// TwinCAT 3 PLC project GW200_plc
// ProgramVersion: 3.1.4024.0
// libraries:
//   Tc2_SerialCom, * (Beckhoff Automation GmbH)
//   Tc2_Standard, * (Beckhoff Automation GmbH)
//   Tc2_System, * (Beckhoff Automation GmbH)
//   Tc2_Utilities, * (Beckhoff Automation GmbH)
//   Tc3_JsonXml, * (Beckhoff Automation GmbH)
//   Tc3_Module, * (Beckhoff Automation GmbH)
// project tree:
//   Base/Alarms/Alarm/ E_ALARM_ACK_TYPE.TcDUT, E_ALARM_STATE.TcDUT, FB_ALARM.TcPOU, TYP_ALARM_CONFIG.TcDUT
//   Base/Alarms/Handler/ FBA_ALARM_HANDLER.TcPOU, FB_ALARM_HANDLER.TcPOU
//   Base/Alarms/ I_ALARM_HANDLER.TcIO, TYP_ALARM_DEVICE_CONFIG.TcDUT
//   Base/Alarms/Repository/ FB_ALARM_INSTANCE.TcPOU, FB_ALARM_REPOSITORY.TcPOU, TYP_ALARM_HISTORY_ENTRY.TcDUT, TYP_VISU_ALARM.TcDUT
//   Base/ BASE.TcPOU
//   Base/Basic/ FB_RS_TRIG.TcPOU
//   Base/DateTime/ FB_DATETIME.TcPOU
//   Base/Files/ FB_FIND_FILES.TcPOU
//   Base/Math/ FC_SCALE.TcPOU, TYP_SCALE_CONF.TcDUT
//   Base/Motion/DC/DcMotor/ FB_DC_MOTOR.TcPOU, TYP_DC_MOTOR_STATUS.TcDUT
//   Base/Motion/DC/DcMotor/Hardware/ TYP_DC_MOTOR_HW.TcDUT, TYP_DC_MOTOR_HW_IN.TcDUT, TYP_DC_MOTOR_HW_OUT.TcDUT
//   Base/Motion/DC/Faulhaber_SC/ FB_FAULHABER_SC.TcPOU, TYP_FAULHABER_SC_CTRL.TcDUT
//   Base/Motion/DC/Faulhaber_SC/Hardware/ TYP_FAULHABER_SC_HW.TcDUT, TYP_FAULHABER_SC_HW_IN.TcDUT, TYP_FAULHABER_SC_HW_OUT.TcDUT
//   Base/Pneumatics/ FB_VALVE_TIMEOUT_ALARM.TcPOU, TYP_VALVE_POS_CONF.TcDUT, TYP_VALVE_POS_HW.TcDUT, TYP_VALVE_TIMEOUT_ALARM_CONF.TcDUT
//   Base/Pneumatics/VacuumGen/ FB_VAC_GEN.TcPOU, TYP_VAC_GEN_ALARM_CONF.TcDUT, TYP_VAC_GEN_CONF.TcDUT, TYP_VAC_GEN_CTRL.TcDUT, TYP_VAC_GEN_STATUS.TcDUT
//   Base/Pneumatics/VacuumGen/Hardware/ TYP_VAC_GEN_HW.TcDUT, TYP_VAC_GEN_HW_IN.TcDUT, TYP_VAC_GEN_HW_OUT.TcDUT
//   Base/Pneumatics/Valve53/ FB_VALVE_53.TcPOU, TYP_VALVE_53_CONF.TcDUT, TYP_VALVE_53_CTRL.TcDUT, TYP_VALVE_53_STATUS.TcDUT
//   Base/Pneumatics/Valve53/Hardware/ TYP_VALVE_53_HW.TcDUT, TYP_VALVE_53_HW_IN.TcDUT, TYP_VALVE_53_HW_OUT.TcDUT
//   Base/Robotics/ TYP_REAL_XYZ.TcDUT
//   Base/Robotics/UR/Profinet/ E_UR_PN_ROBOT_MODE.TcDUT, FB_UR_PN.TcPOU, FB_UR_PN_IO.TcPOU, TYP_HW_UR_PN.TcDUT, TYP_HW_UR_PN_IN.TcDUT, TYP_HW_UR_PN_OUT.TcDUT, TYP_UR_PN_STATE.TcDUT, TYP_UR_PN_TCP.TcDUT
//   Base/Serial/ FB_EL6001_LINE_CTRL.TcPOU, FB_EL6001_RS232.TcPOU, TYP_HW_EL6001.TcDUT, TYP_HW_EL6001_IN.TcDUT, TYP_HW_EL6001_OUT.TcDUT, TYP_SERIAL_DATA.TcDUT
//   Base/Signalling/BannerK50/ FB_BANNER_K50.TcPOU
//   Base/Signalling/BannerK50/Hardware/ TYP_BAN_K50_HW.TcDUT, TYP_BAN_K50_HW_IN.TcDUT, TYP_BAN_K50_HW_OUT.TcDUT
//   Base/Signalling/Lights/ TYP_RYG_TOWER_HW.TcDUT, TYP_RYG_TOWER_HW_OUT.TcDUT
//   Base/Signalling/RGB/ FB_RGB_LED.TcPOU
//   Base/Signalling/RGB/Hardware/ TYP_RGB_LED_CHANNEL.TcDUT, TYP_RGB_LED_CHANNEL_OUT.TcDUT, TYP_RGB_LED_HW.TcDUT
//   Base/States/ FBA_SEQUENCE.TcPOU, FB_SEQUENCE_VISU.TcPOU, FB_STATE_MACHINE.TcPOU
//   Base/String/ FB_STRINGS.TcPOU
//   Base/Tooling/DepragAST11/ TYP_DEPRAG_AST11_HW.TcDUT, TYP_DEPRAG_AST11_HW_IN.TcDUT, TYP_DEPRAG_AST11_HW_OUT.TcDUT
//   Base/Twiddlers/ FC_FLIP_DWORD.TcPOU, FC_FLIP_WORD.TcPOU, FC_GET_BIT_IN_BYTE.TcPOU, FC_MEMCPY_FLIP_WORD.TcPOU, FC_MEMCPY_SWAP_BYTE.TcPOU, FC_MEMCPY_SWAP_WORD.TcPOU, FC_SET_BIT_IN_BYTE.TcPOU
//   Base/Vision/Cognex/3D_L4000/OpcUa/ TYP_HW_L4000_OPC.TcDUT, TYP_HW_L4000_OPC_IN.TcDUT, TYP_HW_L4000_OPC_JOB_CHANGE.TcDUT, TYP_HW_L4000_OPC_JOB_CHANGE_IN.TcDUT, TYP_HW_L4000_OPC_JOB_CHANGE_OUT.TcDUT, TYP_HW_L4000_OPC_OUT.TcDUT
//   Base/Vision/Cognex/3D_L4000/Profinet/ TYP_HW_L4000.TcDUT, TYP_HW_L4000_ACQ_CTRL.TcDUT, TYP_HW_L4000_ACQ_STATUS.TcDUT, TYP_HW_L4000_EXT_CTRL.TcDUT, TYP_HW_L4000_EXT_STATUS.TcDUT, TYP_HW_L4000_IN.TcDUT, TYP_HW_L4000_INSP_CTRL.TcDUT, TYP_HW_L4000_INSP_RESULTS.TcDUT, TYP_HW_L4000_INSP_STATUS.TcDUT, TYP_HW_L4000_OUT.TcDUT
//   Main/ E_MAIN_STATE.TcDUT, E_COLD_START_STATE.TcDUT, MAIN.TcPOU
//   Main/PressureControl/ FB_PRES_CNTRL.TcPOU, gPresCntrl.TcGVL, TYP_PRES_CNTRL_STATUS.TcDUT, TYP_PRES_CNTRL_PARAMETER.TcDUT, TYP_PRES_CNTRL_CONTROL.TcDUT
//   Main/PurgeN2/ E_N2_STATES.TcDUT, FB_N2_DEVICE.TcPOU, FB_PURGE_N2.TcPOU, gPurgeN2.TcGVL, TYP_PURGE_N2_STATUS.TcDUT, TYP_PURGE_N2_PARAMETER.TcDUT, TYP_PURGE_N2_CONTROL.TcDUT
//   / PlcTask.TcTTO
// real-time tasks:
//   TASK PlcTask: cycle T#10ms, priority 20, ADS port 350

CONFIGURATION GW200_plc
    RESOURCE PLC ON TwinCAT3
        TASK PlcTask(INTERVAL := T#10ms, PRIORITY := 20);
        PROGRAM MAIN WITH PlcTask : MAIN;
    END_RESOURCE
END_CONFIGURATION

// ---- Base/Alarms/Alarm/E_ALARM_ACK_TYPE.TcDUT
{attribute 'qualified_only'}
{attribute 'strict'}
TYPE E_ALARM_ACK_TYPE :
(
	ONLY_ACK := 0, // Alarm will clear only after acknowledgement, reset not necessary
	ONLY_RESET := 1, // Alarm will clear only after reset, acknowledgement not necessary
	ACK_AFTER_RESET := 2, // Alarm will clear if acknowledgement is done after reset
	ACK_OR_RESET := 3, // Alarm will clear if reset or acknowledged, whichever comes first
	ACK_AND_RESET := 4 // Alarm will clear if reset and acknowledged, order not important
);
END_TYPE

// ---- Base/Alarms/Alarm/E_ALARM_STATE.TcDUT
{attribute 'qualified_only'}
{attribute 'strict'}
{attribute 'to_string'}
TYPE E_ALARM_STATE :
(
	INACTIVE := 0,
	ACTIVE_UNACK := 1,
	ACTIVE_ACK := 2,
	INACTIVE_UNACK := 4
);
END_TYPE

// ---- Base/Alarms/Alarm/TYP_ALARM_CONFIG.TcDUT
TYPE TYP_ALARM_CONFIG :
STRUCT
	Name : STRING;
	Priority : INT;
	Code : DINT;
	Acknowledge : E_ALARM_ACK_TYPE;
	MultiInstance : BOOL; // Alarm going active again creates new alarm instance
END_STRUCT
END_TYPE

// ---- Base/Alarms/Repository/TYP_ALARM_HISTORY_ENTRY.TcDUT
TYPE TYP_ALARM_HISTORY_ENTRY :
STRUCT
	Timestamp : DT;
	Name : STRING;
	Message : STRING;
	PreviousState : STRING;
	NewState : STRING;
	Code : DINT;
	Priority : INT;
END_STRUCT
END_TYPE

// ---- Base/Alarms/Repository/TYP_VISU_ALARM.TcDUT
TYPE TYP_VISU_ALARM :
STRUCT
	Timestamp : DT;
	Name : STRING;
	Message : STRING;
	State : STRING;
	Code : DINT;
	Priority : INT;
END_STRUCT
END_TYPE

// ---- Base/Alarms/TYP_ALARM_DEVICE_CONFIG.TcDUT
TYPE TYP_ALARM_DEVICE_CONFIG :
STRUCT
	Name : STRING;
	Handler : REFERENCE TO FB_ALARM_HANDLER;
END_STRUCT
END_TYPE

// ---- Base/Math/TYP_SCALE_CONF.TcDUT
TYPE TYP_SCALE_CONF :
STRUCT
	InMin : REAL;
	InMax : REAL;
	OutMin : REAL;
	OutMax : REAL;
END_STRUCT
END_TYPE

// ---- Base/Motion/DC/DcMotor/Hardware/TYP_DC_MOTOR_HW.TcDUT
TYPE TYP_DC_MOTOR_HW :
STRUCT
	In : TYP_DC_MOTOR_HW_IN;
	Out : TYP_DC_MOTOR_HW_OUT;
END_STRUCT
END_TYPE

// ---- Base/Motion/DC/DcMotor/Hardware/TYP_DC_MOTOR_HW_IN.TcDUT
TYPE TYP_DC_MOTOR_HW_IN :
STRUCT
	LimitHP AT %I* : BOOL;
	LimitWP AT %I* : BOOL;
END_STRUCT
END_TYPE

// ---- Base/Motion/DC/DcMotor/Hardware/TYP_DC_MOTOR_HW_OUT.TcDUT
TYPE TYP_DC_MOTOR_HW_OUT :
STRUCT
	Direction AT %Q* : BOOL;
	Run AT %Q* : BOOL;
END_STRUCT
END_TYPE

// ---- Base/Motion/DC/DcMotor/TYP_DC_MOTOR_STATUS.TcDUT
TYPE TYP_DC_MOTOR_STATUS :
STRUCT
	ReachedHP : BOOL;
	ReachedWP : BOOL;
END_STRUCT
END_TYPE

// ---- Base/Motion/DC/Faulhaber_SC/Hardware/TYP_FAULHABER_SC_HW.TcDUT
TYPE TYP_FAULHABER_SC_HW :
STRUCT
	In : TYP_FAULHABER_SC_HW_IN;
	Out : TYP_FAULHABER_SC_HW_OUT;
END_STRUCT
END_TYPE

// ---- Base/Motion/DC/Faulhaber_SC/Hardware/TYP_FAULHABER_SC_HW_IN.TcDUT
TYPE TYP_FAULHABER_SC_HW_IN :
STRUCT
	Fault AT %I*: BOOL;
END_STRUCT
END_TYPE

// ---- Base/Motion/DC/Faulhaber_SC/Hardware/TYP_FAULHABER_SC_HW_OUT.TcDUT
TYPE TYP_FAULHABER_SC_HW_OUT :
STRUCT
	Speed AT %Q*: INT;
	Direction AT %Q*: BOOL;
END_STRUCT
END_TYPE

// ---- Base/Motion/DC/Faulhaber_SC/TYP_FAULHABER_SC_CTRL.TcDUT
TYPE TYP_FAULHABER_SC_CTRL :
STRUCT	
	Enable : BOOL; // Enable action
	Run : BOOL; // Run motor
	Speed : INT; // Setpoint speed
END_STRUCT
END_TYPE

// ---- Base/Pneumatics/TYP_VALVE_POS_CONF.TcDUT
TYPE TYP_VALVE_POS_CONF :
STRUCT
	Sensorless : BOOL; (* no sensor, reached status after SensorlessDelay *)
	SensorlessDelay : TIME; (* delay for reached status in sensorless mode *)
	Permanent : BOOL := TRUE; // Output stays on after reaching position
	Timeout : TYP_VALVE_TIMEOUT_ALARM_CONF;
END_STRUCT
END_TYPE

// ---- Base/Pneumatics/TYP_VALVE_POS_HW.TcDUT
TYPE TYP_VALVE_POS_HW :
STRUCT
	ReachedHP AT %I* : BOOL;
	ReachedWP AT %I* : BOOL;
END_STRUCT
END_TYPE

// ---- Base/Pneumatics/TYP_VALVE_TIMEOUT_ALARM_CONF.TcDUT
TYPE TYP_VALVE_TIMEOUT_ALARM_CONF :
STRUCT
	Enable : BOOL := TRUE; // Alarm enabled
	Delay : TIME := T#10S; // Delay before alarm is activated
END_STRUCT
END_TYPE

// ---- Base/Pneumatics/VacuumGen/Hardware/TYP_VAC_GEN_HW.TcDUT
TYPE TYP_VAC_GEN_HW :
STRUCT
	In : TYP_VAC_GEN_HW_IN;
	Out : TYP_VAC_GEN_HW_OUT;
END_STRUCT
END_TYPE

// ---- Base/Pneumatics/VacuumGen/Hardware/TYP_VAC_GEN_HW_IN.TcDUT
TYPE TYP_VAC_GEN_HW_IN :
STRUCT
	ReachedVac AT %I* : BOOL;
END_STRUCT
END_TYPE

// ---- Base/Pneumatics/VacuumGen/Hardware/TYP_VAC_GEN_HW_OUT.TcDUT
TYPE TYP_VAC_GEN_HW_OUT :
STRUCT
	EnableVac AT %Q* : BOOL;
	ReleaseVac AT %Q* : BOOL;
END_STRUCT
END_TYPE

// ---- Base/Pneumatics/VacuumGen/TYP_VAC_GEN_ALARM_CONF.TcDUT
TYPE TYP_VAC_GEN_ALARM_CONF :
STRUCT
	Enable : BOOL := TRUE;
	Timeout : TIME := T#4S;
END_STRUCT
END_TYPE

// ---- Base/Pneumatics/VacuumGen/TYP_VAC_GEN_CONF.TcDUT
TYPE TYP_VAC_GEN_CONF :
STRUCT
	Permanent : BOOL := TRUE; // Holds output even after reaching vacuum
	Alarm : TYP_VAC_GEN_ALARM_CONF;
END_STRUCT
END_TYPE

// ---- Base/Pneumatics/VacuumGen/TYP_VAC_GEN_CTRL.TcDUT
TYPE TYP_VAC_GEN_CTRL :
STRUCT
	Enable : BOOL := TRUE; // Enable vacuum gen control
	EnableActivate : BOOL := TRUE; // Enable vacuum activation
	EnableRelease : BOOL := TRUE; // Enable release activation
	ServiceEnable : BOOL;
	ServiceActivate : BOOL;
	ServiceRelease : BOOL;
END_STRUCT
END_TYPE

// ---- Base/Pneumatics/VacuumGen/TYP_VAC_GEN_STATUS.TcDUT
TYPE TYP_VAC_GEN_STATUS :
STRUCT
	ReachedVac : BOOL;
	Error : BOOL;
END_STRUCT
END_TYPE

// ---- Base/Pneumatics/Valve53/Hardware/TYP_VALVE_53_HW.TcDUT
TYPE TYP_VALVE_53_HW :
STRUCT
	In : TYP_VALVE_53_HW_IN;
	Out : TYP_VALVE_53_HW_OUT;
END_STRUCT
END_TYPE

// ---- Base/Pneumatics/Valve53/Hardware/TYP_VALVE_53_HW_IN.TcDUT
TYPE TYP_VALVE_53_HW_IN :
STRUCT
	ReachedHP AT %I* : BOOL;
	ReachedWP AT %I* : BOOL;
END_STRUCT
END_TYPE

// ---- Base/Pneumatics/Valve53/Hardware/TYP_VALVE_53_HW_OUT.TcDUT
TYPE TYP_VALVE_53_HW_OUT :
STRUCT
	CmdHP AT %Q* : BOOL;
	CmdWP AT %Q* : BOOL;
END_STRUCT
END_TYPE

// ---- Base/Pneumatics/Valve53/TYP_VALVE_53_CONF.TcDUT
TYPE TYP_VALVE_53_CONF :
STRUCT
	HP : TYP_VALVE_POS_CONF;
	WP : TYP_VALVE_POS_CONF;
	HP_WP : TYP_VALVE_TIMEOUT_ALARM_CONF; // Alarm for both HP and WP sensors active
END_STRUCT
END_TYPE

// ---- Base/Pneumatics/Valve53/TYP_VALVE_53_CTRL.TcDUT
TYPE TYP_VALVE_53_CTRL :
STRUCT
	Enable : BOOL := TRUE; (* Enable movement in auto mode *)
	EnableHP : BOOL := TRUE; (* Allow movement to HP *)
	EnableWP : BOOL := TRUE; (* Allow movement to WP *)
	ServiceEnable : BOOL; (* Enable movement in Service Mode NB!! This ignores all other enable/disable commands *)
	ServiceHP : BOOL; (* Command movement to Home Position NB!! This ignores all other enable/disable commands *)
	ServiceWP : BOOL; (* Command movement to Wome Position NB!! This ignores all other enable/disable commands *)
	BlockOutputs : BOOL; // Do not allow to switch outputs
END_STRUCT
END_TYPE

// ---- Base/Pneumatics/Valve53/TYP_VALVE_53_STATUS.TcDUT
TYPE TYP_VALVE_53_STATUS :
STRUCT
	ReachedHP : BOOL;
	ReachedWP : BOOL;
	Error : BOOL;
END_STRUCT
END_TYPE

// ---- Base/Robotics/TYP_REAL_XYZ.TcDUT
TYPE TYP_REAL_XYZ :
STRUCT
	X : REAL;
	Y : REAL;
	Z : REAL;
END_STRUCT
END_TYPE

// ---- Base/Robotics/UR/Profinet/E_UR_PN_ROBOT_MODE.TcDUT
{attribute 'qualified_only'}
//{attribute 'strict'}
{attribute 'to_string'}
TYPE E_UR_PN_ROBOT_MODE :
(
	DISCONNECTED := 0,
	CONFIRM_SAFETY := 1,
	BOOTING := 2,
	POWER_OFF := 3,
	POWER_ON := 4,
	IDLE := 5,
	BACKDRIVE := 6,
	RUNNING := 7
);
END_TYPE

// ---- Base/Robotics/UR/Profinet/TYP_HW_UR_PN.TcDUT
TYPE TYP_HW_UR_PN :
STRUCT
	In : TYP_HW_UR_PN_IN;
	Out : TYP_HW_UR_PN_OUT;
END_STRUCT
END_TYPE

// ---- Base/Robotics/UR/Profinet/TYP_HW_UR_PN_IN.TcDUT
TYPE TYP_HW_UR_PN_IN :
STRUCT
	T2OURState AT %I*: ARRAY[0..31] OF BYTE;
	T2OURIO AT %I*: ARRAY[0..67] OF BYTE;
	T2OURJoints AT %I*: ARRAY[0..103] OF BYTE;
	T2OURTCP AT %I*: ARRAY[0..75] OF BYTE;
	T2OURBitReg AT %I*: ARRAY[0..7] OF BYTE;
	T2OURIntReg AT %I*: ARRAY[0..95] OF BYTE;
	T2OURFloatReg AT %I*: ARRAY[0..95] OF BYTE;
END_STRUCT
END_TYPE

// ---- Base/Robotics/UR/Profinet/TYP_HW_UR_PN_OUT.TcDUT
TYPE TYP_HW_UR_PN_OUT :
STRUCT
	O2TURIO AT %Q*: ARRAY[0..23] OF BYTE;
	O2TURGenReg1 AT %Q*: ARRAY[0..99] OF BYTE;
	O2TURGenReg2 AT %Q*: ARRAY[0..99] OF BYTE;
END_STRUCT
END_TYPE

// ---- Base/Robotics/UR/Profinet/TYP_UR_PN_STATE.TcDUT
TYPE TYP_UR_PN_STATE :
STRUCT
	MajVersion : USINT; // Controller major version
	MinVersion : USINT; // Controller minor version
	RobotMode : E_UR_PN_ROBOT_MODE;
	RTMd : UINT; // Real time machine days
	RTMh : UINT; // Real time machine hours
	RTMm : UINT; // Real time machine days
	RTMs : UINT; // Real time machine days
	RTMms : UINT; // Real time machine milliseconds
	Power : BOOL;
	ProgramRunning : BOOL;
	PowerButton : BOOL;
	TeachButton : BOOL;
	RobotCurrent : REAL; // Current power consumption A
	NormalMode: BOOL;
	ReducedMode: BOOL;
	ProtectiveStopped: BOOL;
	RecoveryMode: BOOL;
	SafeguardStop: BOOL;
	SystemEmergencyStopped: BOOL;
	RobotEmergencyStopped: BOOL;
	EmergencyStopped: BOOL;
	Violation: BOOL;
	Faulted: BOOL;
	SafetyStopped: BOOL;
END_STRUCT
END_TYPE

// ---- Base/Robotics/UR/Profinet/TYP_UR_PN_TCP.TcDUT
TYPE TYP_UR_PN_TCP :
STRUCT
	Position : TYP_REAL_XYZ;
	PositionR : TYP_REAL_XYZ;
	Velocity : TYP_REAL_XYZ;
	VelocityR : TYP_REAL_XYZ;
	Force : TYP_REAL_XYZ;
	Torque : TYP_REAL_XYZ;
	ForceScalar : REAL;
END_STRUCT
END_TYPE

// ---- Base/Serial/TYP_HW_EL6001.TcDUT
TYPE TYP_HW_EL6001 :
STRUCT
	In : TYP_HW_EL6001_IN;
	Out : TYP_HW_EL6001_OUT;
END_STRUCT
END_TYPE

// ---- Base/Serial/TYP_HW_EL6001_IN.TcDUT
TYPE TYP_HW_EL6001_IN :
STRUCT
	COM AT %I*: KL6InData22B;
END_STRUCT
END_TYPE

// ---- Base/Serial/TYP_HW_EL6001_OUT.TcDUT
TYPE TYP_HW_EL6001_OUT :
STRUCT
	COM AT %Q* : KL6OutData22B;
END_STRUCT
END_TYPE

// ---- Base/Serial/TYP_SERIAL_DATA.TcDUT
TYPE TYP_SERIAL_DATA :
STRUCT
	RxData : COMbuffer;
	TxData : COMbuffer;
END_STRUCT
END_TYPE

// ---- Base/Signalling/BannerK50/Hardware/TYP_BAN_K50_HW.TcDUT
TYPE TYP_BAN_K50_HW :
STRUCT
	In : TYP_BAN_K50_HW_IN;
	Out : TYP_BAN_K50_HW_OUT;
END_STRUCT
END_TYPE

// ---- Base/Signalling/BannerK50/Hardware/TYP_BAN_K50_HW_IN.TcDUT
TYPE TYP_BAN_K50_HW_IN :
STRUCT
	ButtonPressed AT %I* : BOOL;
END_STRUCT
END_TYPE

// ---- Base/Signalling/BannerK50/Hardware/TYP_BAN_K50_HW_OUT.TcDUT
TYPE TYP_BAN_K50_HW_OUT :
STRUCT
	Red AT %Q* : BOOL;
	Yellow AT %Q* : BOOL;
	Green AT %Q* : BOOL;
END_STRUCT
END_TYPE

// ---- Base/Signalling/Lights/TYP_RYG_TOWER_HW.TcDUT
TYPE TYP_RYG_TOWER_HW :
STRUCT
	Out : TYP_RYG_TOWER_HW_OUT;
END_STRUCT
END_TYPE

// ---- Base/Signalling/Lights/TYP_RYG_TOWER_HW_OUT.TcDUT
TYPE TYP_RYG_TOWER_HW_OUT :
STRUCT
	Red AT %Q* : BOOL;
	Yellow AT %Q* : BOOL;
	Green AT %Q* : BOOL;
END_STRUCT
END_TYPE

// ---- Base/Signalling/RGB/Hardware/TYP_RGB_LED_CHANNEL.TcDUT
TYPE TYP_RGB_LED_CHANNEL :
STRUCT
	Out : TYP_RGB_LED_CHANNEL_OUT;
END_STRUCT
END_TYPE

// ---- Base/Signalling/RGB/Hardware/TYP_RGB_LED_CHANNEL_OUT.TcDUT
TYPE TYP_RGB_LED_CHANNEL_OUT :
STRUCT
	PWM AT %Q* : INT;
END_STRUCT
END_TYPE

// ---- Base/Signalling/RGB/Hardware/TYP_RGB_LED_HW.TcDUT
TYPE TYP_RGB_LED_HW :
STRUCT
	Red : TYP_RGB_LED_CHANNEL;
	Green : TYP_RGB_LED_CHANNEL;
	Blue : TYP_RGB_LED_CHANNEL;
END_STRUCT
END_TYPE

// ---- Base/Tooling/DepragAST11/TYP_DEPRAG_AST11_HW.TcDUT
TYPE TYP_DEPRAG_AST11_HW :
STRUCT
	In : TYP_DEPRAG_AST11_HW_IN;
	Out : TYP_DEPRAG_AST11_HW_OUT;
END_STRUCT
END_TYPE

// ---- Base/Tooling/DepragAST11/TYP_DEPRAG_AST11_HW_IN.TcDUT
TYPE TYP_DEPRAG_AST11_HW_IN :
STRUCT
	Ready AT %I*: BOOL;
	OK AT %I*: BOOL;
	NOK AT %I*: BOOL;
END_STRUCT
END_TYPE

// ---- Base/Tooling/DepragAST11/TYP_DEPRAG_AST11_HW_OUT.TcDUT
TYPE TYP_DEPRAG_AST11_HW_OUT :
STRUCT
	Start AT %Q*: BOOL;
END_STRUCT
END_TYPE

// ---- Base/Vision/Cognex/3D_L4000/OpcUa/TYP_HW_L4000_OPC.TcDUT
TYPE TYP_HW_L4000_OPC :
STRUCT
	LoadJob : TYP_HW_L4000_OPC_JOB_CHANGE;
	In : TYP_HW_L4000_OPC_IN;
	Out : TYP_HW_L4000_OPC_OUT;
END_STRUCT
END_TYPE

// ---- Base/Vision/Cognex/3D_L4000/OpcUa/TYP_HW_L4000_OPC_IN.TcDUT
TYPE TYP_HW_L4000_OPC_IN :
STRUCT
	Result AT %I* : ARRAY[1..43] OF REAL;
	Online AT %I* : BOOL;
	ActiveJob AT %I* : STRING;
END_STRUCT
END_TYPE

// ---- Base/Vision/Cognex/3D_L4000/OpcUa/TYP_HW_L4000_OPC_JOB_CHANGE.TcDUT
TYPE TYP_HW_L4000_OPC_JOB_CHANGE :
STRUCT
	In : TYP_HW_L4000_OPC_JOB_CHANGE_IN;
	Out : TYP_HW_L4000_OPC_JOB_CHANGE_OUT;
END_STRUCT
END_TYPE

// ---- Base/Vision/Cognex/3D_L4000/OpcUa/TYP_HW_L4000_OPC_JOB_CHANGE_IN.TcDUT
TYPE TYP_HW_L4000_OPC_JOB_CHANGE_IN :
STRUCT
	ErrorID AT %I* : DINT;
	Done AT %I* : BOOL;
	Busy AT %I* : BOOL;
	Error AT %I* : BOOL;
END_STRUCT
END_TYPE

// ---- Base/Vision/Cognex/3D_L4000/OpcUa/TYP_HW_L4000_OPC_JOB_CHANGE_OUT.TcDUT
TYPE TYP_HW_L4000_OPC_JOB_CHANGE_OUT :
STRUCT
	Execute AT %Q* : BOOL;
	Filename AT %Q* : STRING;
END_STRUCT
END_TYPE

// ---- Base/Vision/Cognex/3D_L4000/OpcUa/TYP_HW_L4000_OPC_OUT.TcDUT
TYPE TYP_HW_L4000_OPC_OUT :
STRUCT
	WriteEnable AT %Q* : BOOL;
	Online AT %Q* : BOOL;
END_STRUCT
END_TYPE

// ---- Base/Vision/Cognex/3D_L4000/Profinet/TYP_HW_L4000.TcDUT
TYPE TYP_HW_L4000 :
STRUCT
	In : TYP_HW_L4000_IN;
	Out : TYP_HW_L4000_OUT;
END_STRUCT
END_TYPE

// ---- Base/Vision/Cognex/3D_L4000/Profinet/TYP_HW_L4000_ACQ_CTRL.TcDUT
TYPE TYP_HW_L4000_ACQ_CTRL :
STRUCT
	AcqTriggerEnable AT %Q* : BOOL;
	AcqTrigger AT %Q* : BOOL;
	ClearExposureComplete AT %Q* : BOOL;
	SetPauseOfOnline AT %Q* : BOOL;
END_STRUCT
END_TYPE

// ---- Base/Vision/Cognex/3D_L4000/Profinet/TYP_HW_L4000_ACQ_STATUS.TcDUT
TYPE TYP_HW_L4000_ACQ_STATUS :
STRUCT
	AcqTriggerReady AT %I* : BOOL;
	AcqTriggerAcknowledge AT %I* : BOOL;
	ExposureComplete AT %I* : BOOL;
	AcqError AT %I* : BOOL;
	Paused AT %I* : BOOL;
	Online AT %I* : BOOL;
	AcqID AT %I* : UINT;
END_STRUCT
END_TYPE

// ---- Base/Vision/Cognex/3D_L4000/Profinet/TYP_HW_L4000_EXT_CTRL.TcDUT
TYPE TYP_HW_L4000_EXT_CTRL :
STRUCT
	Trigger AT %Q* : ARRAY[0..7] OF BOOL;
END_STRUCT
END_TYPE

// ---- Base/Vision/Cognex/3D_L4000/Profinet/TYP_HW_L4000_EXT_STATUS.TcDUT
TYPE TYP_HW_L4000_EXT_STATUS :
STRUCT
	Acknowledge AT %I* : ARRAY[0..7] OF BOOL;
END_STRUCT
END_TYPE

// ---- Base/Vision/Cognex/3D_L4000/Profinet/TYP_HW_L4000_IN.TcDUT
TYPE TYP_HW_L4000_IN :
STRUCT
	AcqStatus : TYP_HW_L4000_ACQ_STATUS;
	InspStatus : TYP_HW_L4000_INSP_STATUS;
	CommandResult AT %I* : UINT;
	ExternalEvent : TYP_HW_L4000_EXT_STATUS;
	InspResults : TYP_HW_L4000_INSP_RESULTS;
END_STRUCT
END_TYPE

// ---- Base/Vision/Cognex/3D_L4000/Profinet/TYP_HW_L4000_INSP_CTRL.TcDUT
TYPE TYP_HW_L4000_INSP_CTRL :
STRUCT
	EnableResultsBuffering AT %Q* : BOOL;
	AckInspectionResults AT %Q* : BOOL;
	SetUserData AT %Q* : BOOL;
	ExecuteCommand AT %Q* : BOOL;
	ClearError AT %Q* : BOOL;
END_STRUCT
END_TYPE

// ---- Base/Vision/Cognex/3D_L4000/Profinet/TYP_HW_L4000_INSP_RESULTS.TcDUT
TYPE TYP_HW_L4000_INSP_RESULTS :
STRUCT
	InspectionID AT %I* : UINT;
	InspectionResultCode AT %I* : UINT;
	Results AT %I* : ARRAY[0..63] OF BYTE;
END_STRUCT
END_TYPE

// ---- Base/Vision/Cognex/3D_L4000/Profinet/TYP_HW_L4000_INSP_STATUS.TcDUT
TYPE TYP_HW_L4000_INSP_STATUS :
STRUCT
	SystemReady AT %I* : BOOL;
	InspectionCompleted AT %I* : BOOL;
	ResultsBufferOverrun AT %I* : BOOL;
	ResultsValid AT %I* : BOOL;
	CommandExecuting AT %I* : BOOL;
	CommandCompleted AT %I* : BOOL;
	CommandFailed AT %I* : BOOL;
	SetUserDataAcknowledge AT %I* : BOOL;
	ResultsPassed AT %I* : BOOL;
	Error AT %I* : BOOL;
	ErrorID AT %I* : UINT;
END_STRUCT
END_TYPE

// ---- Base/Vision/Cognex/3D_L4000/Profinet/TYP_HW_L4000_OUT.TcDUT
TYPE TYP_HW_L4000_OUT :
STRUCT
	AcqCtrl : TYP_HW_L4000_ACQ_CTRL;
	InspCtrl : TYP_HW_L4000_INSP_CTRL;
	CommandID AT %Q* : UINT;
	ExternalEvent : TYP_HW_L4000_EXT_CTRL;
	UserData AT %Q* : ARRAY[0..63] OF BYTE;
END_STRUCT
END_TYPE

// ---- Main/E_MAIN_STATE.TcDUT
{attribute 'qualified_only'}
{attribute 'strict'}
TYPE E_MAIN_STATE :
(
	NULL := 0,
	IDLE,
	COLD_START,
	HOT_START,
	SHUT_DOWN,
	PRODUCTION,
	HOT_STANDBY,
	COLD_STANDBY
);
END_TYPE

// ---- Main/E_COLD_START_STATE.TcDUT
{attribute 'qualified_only'}
{attribute 'strict'}
TYPE E_COLD_START_STATE :
(
	NULL := 0,
	N2_PURGE,
	TEMPERATURE,	
	PRESSURISE,
	H2_PURGE
);
END_TYPE

// ---- Main/PressureControl/TYP_PRES_CNTRL_STATUS.TcDUT
TYPE TYP_PRES_CNTRL_STATUS :
STRUCT
	Done : BOOL;
	Executing: BOOL;
	Error : BOOL;
END_STRUCT
END_TYPE

// ---- Main/PressureControl/TYP_PRES_CNTRL_PARAMETER.TcDUT
TYPE TYP_PRES_CNTRL_PARAMETER :
STRUCT
	SetPoint : REAL;
END_STRUCT
END_TYPE

// ---- Main/PressureControl/TYP_PRES_CNTRL_CONTROL.TcDUT
TYPE TYP_PRES_CNTRL_CONTROL :
STRUCT
	Execute : BOOL;
END_STRUCT
END_TYPE

// ---- Main/PurgeN2/E_N2_STATES.TcDUT
{attribute 'qualified_only'}
{attribute 'strict'}
TYPE E_N2_STATES :
(
	STATE1,
	STATE2,
	STATE3
);
END_TYPE

// ---- Main/PurgeN2/TYP_PURGE_N2_STATUS.TcDUT
TYPE TYP_PURGE_N2_STATUS :
STRUCT
	Done : BOOL;
	Executing: BOOL;
	Error : BOOL;
END_STRUCT
END_TYPE

// ---- Main/PurgeN2/TYP_PURGE_N2_PARAMETER.TcDUT
TYPE TYP_PURGE_N2_PARAMETER :
STRUCT
	NoPurge : INT;
END_STRUCT
END_TYPE

// ---- Main/PurgeN2/TYP_PURGE_N2_CONTROL.TcDUT
TYPE TYP_PURGE_N2_CONTROL :
STRUCT
	Execute : BOOL;
END_STRUCT
END_TYPE

// ---- Main/PressureControl/gPresCntrl.TcGVL
{attribute 'qualified_only'}
VAR_GLOBAL
	Control : TYP_PRES_CNTRL_CONTROL;
	Parameter : TYP_PRES_CNTRL_PARAMETER;
	Status : TYP_PRES_CNTRL_STATUS;
END_VAR

// ---- Main/PurgeN2/gPurgeN2.TcGVL
{attribute 'qualified_only'}
VAR_GLOBAL
	Control: TYP_PURGE_N2_CONTROL;
	Parameter : TYP_PURGE_N2_PARAMETER;
	Status : TYP_PURGE_N2_STATUS;
END_VAR

// ---- Base/Alarms/I_ALARM_HANDLER.TcIO
INTERFACE I_ALARM_HANDLER

METHOD RegisterAlarm : REFERENCE TO FBA_ALARM_HANDLER
VAR_INPUT
	Alarm : REFERENCE TO FB_ALARM;
	Prefix : STRING := '';
	Update : BOOL := TRUE;
END_VAR
END_METHOD

END_INTERFACE

// ---- Main/MAIN.TcPOU
PROGRAM MAIN
VAR
	//State machines
	fbMainState : FB_STATE_MACHINE;
	fbColdStartState : FB_STATE_MACHINE;
	eMainState : E_MAIN_STATE;
	eColdStartState : E_COLD_START_STATE;
	//Alarm handler
	fbAlarmRepository : FB_ALARM_REPOSITORY;
	fbMainHandler : FB_ALARM_HANDLER;
	fbColdStartHandler : FB_ALARM_HANDLER;
	fbAlarms : ARRAY[0..99] OF FB_ALARM_INSTANCE;
	fbVisuAlarms : ARRAY[0..99] OF TYP_VISU_ALARM;
	fbEmStopAlarm : FB_ALARM;
	//Control loops and function blocks
	fbPurgeN2 : FB_PURGE_N2;
	fbPresCntrl : FB_PRES_CNTRL;
	
	bTestalarm : BOOL;
	bTestReset : BOOL;
	bTestAcknowledge : BOOL;
	
	getZone : FB_LocalSystemTime;
END_VAR

//Alarm function blocks
fbAlarmRepository(Alarms := fbAlarms, VisuAlarms := fbVisuAlarms);
fbMainHandler(Prefix := 'MAIN', Repository := fbAlarmRepository);
fbColdStartHandler(Prefix := 'COLD_START', Repository := fbAlarmRepository);

fbEmStopAlarm.Config.Acknowledge := E_ALARM_ACK_TYPE.ACK_AND_RESET;
fbEmStopAlarm.Config.Name := 'EMERGENCY_STOP_ACTIVATED';
fbEmStopAlarm.Config.Priority := 3;
fbEmStopAlarm.Config.Code := 0001;
fbEmStopAlarm(Handler := fbMainHandler);

//Control loops, control functionblocks
fbPurgeN2(AlarmRepository := fbAlarmRepository, Control := gPurgeN2.Control, Parameter := gPurgeN2.Parameter, Status => gPurgeN2.Status);
fbPresCntrl(Control := gPresCntrl.Control, Parameter := gPresCntrl.Parameter, Status => gPresCntrl.Status);

//Example how alarms work
IF bTestalarm THEN
	fbEmStopAlarm.Activate();
ELSIF bTestReset THEN
	fbEmStopAlarm.Reset();
ELSIF bTestAcknowledge THEN
	fbEmStopAlarm.Acknowledge();
END_IF

CASE fbMainState.CurrentState OF //Main state machine
	E_MAIN_STATE.IDLE:
	 //
	E_MAIN_STATE.COLD_START: //Cold start state
		CASE fbColdStartState.CurrentState OF
			E_COLD_START_STATE.N2_PURGE: //Nitorgen purge state
				IF fbColdStartState._firstCycle THEN
					gPurgeN2.Parameter.NoPurge := 5;
					gPurgeN2.Control.Execute := TRUE;
					gPresCntrl.Parameter.SetPoint := 2.0;
					gPresCntrl.Control.Execute := TRUE;
				ELSIF NOT fbColdStartState.ChangePending THEN
					IF gPurgeN2.Status.Done THEN
						fbColdStartState.ChangeState(E_COLD_START_STATE.TEMPERATURE);
					END_IF
				END_IF	
			E_COLD_START_STATE.TEMPERATURE:
				//
			E_COLD_START_STATE.PRESSURISE:
				//
			E_COLD_START_STATE.H2_PURGE:
				//
		END_CASE	
	
	E_MAIN_STATE.HOT_STANDBY:
		//
	E_MAIN_STATE.PRODUCTION:
		//
	E_MAIN_STATE.COLD_STANDBY:
		//
	E_MAIN_STATE.HOT_START:
		//
	E_MAIN_STATE.SHUT_DOWN:
		//
END_CASE

getZone();

fbMainState(State := eMainState, AlarmHandler := fbMainHandler, StateAsString := TO_STRING(eMainState));
fbColdStartState(State := eColdStartState, AlarmHandler := fbColdStartHandler, StateAsString := TO_STRING(eColdStartState));

END_PROGRAM

// ---- Base/States/FB_STATE_MACHINE.TcPOU
FUNCTION_BLOCK FB_STATE_MACHINE
VAR_IN_OUT
	State : INT;
	AlarmHandler : FB_ALARM_HANDLER;
END_VAR
VAR_INPUT
	StateAsString : STRING;
	DebugMode : BOOL;
	DebugNext : BOOL;
	StopAllowed : BOOL;
	Timeout : TIME;
END_VAR
VAR_OUTPUT
	CurrentState : INT;
	_firstCycle : BOOL := TRUE;
	StateChangeTime : TIME := TIME();
	Running : BOOL;
	Stopped : BOOL;
	StopRequested : BOOL;
	PreviousState : INT;
END_VAR
VAR
	_changePending : BOOL;
	DelayStart : TIME;
	ChangeDelay : TIME;
	NewState : INT;
	NextState : INT;
	TimeoutAlarm : FB_ALARM;
END_VAR

IF NOT DebugMode THEN
	DebugNext := FALSE;
END_IF;

IF Running AND StopRequested AND StopAllowed THEN
	Running := FALSE;
	Stopped := TRUE;
	StopRequested := FALSE;
END_IF;

IF NewState <> CurrentState AND (NOT DebugMode OR DebugNext) AND Running THEN
	PreviousState := CurrentState;
	CurrentState := NewState;
	StateChangeTime := TIME();
	_firstCycle := TRUE;
	DebugNext := FALSE;
	
	Timeout := T#0S;
	DelayStart := T#0S;
	ChangeDelay := T#0S;
	_changePending := FALSE;
	NextState := 0;
ELSE
	_firstCycle := FALSE;
END_IF;

IF _changePending AND TIME() >= (DelayStart + ChangeDelay) THEN
	THIS^.NewState := NextState;
END_IF;

IF Timeout > T#0S AND THIS^.GetElapsedTime() > Timeout  THEN
	IF NOT TimeoutAlarm.IsActive THEN
		TimeoutAlarm.Config.Name := CONCAT(StateAsString, '*TIMEOUT_ALARM');
		TimeoutAlarm.Activate();
	END_IF;
END_IF;

TimeoutAlarm.Config.Acknowledge := E_ALARM_ACK_TYPE.ONLY_ACK;
TimeoutAlarm.Config.MultiInstance := TRUE;
TimeoutAlarm(Handler := AlarmHandler);

State := CurrentState;

StopAllowed := FALSE;

PROPERTY PUBLIC ChangePending : BOOL
GET
ChangePending := THIS^._changePending;
END_GET
END_PROPERTY

METHOD ChangeState : REFERENCE TO FB_STATE_MACHINE
VAR_INPUT
	State : INT;
END_VAR
IF NOT _changePending AND THIS^.Running THEN
	_changePending := TRUE;
	NextState := State;
END_IF;

ChangeState REF= THIS^;
END_METHOD

METHOD ChangeStateAfterDelay : REFERENCE TO FB_STATE_MACHINE
VAR_INPUT
	State : INT;
	Delay : TIME;
END_VAR
IF NOT _changePending AND THIS^.Running THEN
	_changePending := TRUE;
	NextState := State;
	DelayStart := TIME();
	ChangeDelay := Delay;
END_IF;

ChangeStateAfterDelay REF= THIS^;
END_METHOD

PROPERTY PUBLIC FirstCycle : BOOL
GET
FirstCycle := _firstCycle AND Running;
END_GET
END_PROPERTY

METHOD PUBLIC GetElapsedTime : TIME
VAR_INPUT
END_VAR
GetElapsedTime := TIME() - StateChangeTime;
END_METHOD

METHOD PUBLIC Reset : REFERENCE TO FB_STATE_MACHINE
VAR_INPUT
END_VAR
THIS^.CurrentState := 0;
THIS^.NewState := 0;
THIS^._firstCycle := TRUE;
THIS^.StateChangeTime := TIME();
THIS^._changePending := FALSE;
THIS^.DelayStart := T#0S;
THIS^.ChangeDelay := T#0S;
THIS^.NextState := 0;
THIS^.Running := FALSE;
THIS^.Stopped := FALSE;
THIS^.StopRequested := FALSE;

Reset REF= THIS^;
END_METHOD

{attribute 'TcRpcEnable'}
METHOD PUBLIC Start : REFERENCE TO FB_STATE_MACHINE
VAR_INPUT
END_VAR
THIS^.Running := TRUE;
THIS^.StopRequested := FALSE;

Start REF= THIS^;
END_METHOD

{attribute 'TcRpcEnable'}
METHOD PUBLIC Stop : REFERENCE TO FB_STATE_MACHINE
VAR_INPUT
END_VAR
THIS^.StopRequested := TRUE;

Stop REF= THIS^;
END_METHOD

END_FUNCTION_BLOCK

// ---- Base/Alarms/Handler/FB_ALARM_HANDLER.TcPOU
FUNCTION_BLOCK PUBLIC FB_ALARM_HANDLER EXTENDS FBA_ALARM_HANDLER
VAR_IN_OUT
	Repository : FBA_ALARM_HANDLER;
END_VAR
VAR_INPUT
	Prefix : STRING;
END_VAR
VAR_OUTPUT
END_VAR
VAR
END_VAR

METHOD RegisterAlarm : REFERENCE TO FBA_ALARM_HANDLER
VAR_INPUT
	Alarm	: REFERENCE TO FB_ALARM;
	Prefix	: STRING := '';
	Update : BOOL := TRUE;
END_VAR
VAR
	TempString : STRING := '';
END_VAR
{warning disable C0371}

// Checking the VAR_IN_OUT reference, leave the current method in case of invalid reference
IF NOT __ISVALIDREF(THIS^.Repository) THEN
     RETURN;
END_IF


IF THIS^.Prefix <> '' THEN
	TempString := CONCAT(THIS^.Prefix, '*');
END_IF;

TempString := CONCAT(TempString, Prefix);
THIS^.Repository.RegisterAlarm(Alarm := Alarm, Prefix := TempString, Update := TRUE);

RegisterAlarm REF= THIS^;
END_METHOD

END_FUNCTION_BLOCK

// ---- Base/Alarms/Handler/FBA_ALARM_HANDLER.TcPOU
FUNCTION_BLOCK PUBLIC ABSTRACT FBA_ALARM_HANDLER IMPLEMENTS I_ALARM_HANDLER
VAR_INPUT
END_VAR
VAR_OUTPUT
END_VAR
VAR
END_VAR

METHOD ABSTRACT RegisterAlarm : REFERENCE TO FBA_ALARM_HANDLER
VAR_INPUT
	Alarm	: REFERENCE TO FB_ALARM;
	Prefix	: STRING := '';
	Update : BOOL := TRUE;
END_VAR
END_METHOD

END_FUNCTION_BLOCK

// ---- Base/Alarms/Alarm/FB_ALARM.TcPOU
FUNCTION_BLOCK PUBLIC FB_ALARM
VAR_IN_OUT
	Handler : FB_ALARM_HANDLER;
END_VAR
VAR_INPUT
	Config : TYP_ALARM_CONFIG;
END_VAR
VAR_OUTPUT
	State : E_ALARM_STATE;
END_VAR

METHOD PUBLIC Acknowledge : REFERENCE TO FB_ALARM
VAR_INPUT
END_VAR
VAR
	PreviousState : E_ALARM_STATE;
END_VAR
{warning disable C0371}

// Checking the VAR_IN_OUT reference, leave the current method in case of invalid reference
IF NOT __ISVALIDREF(THIS^.Handler) THEN
     RETURN;
END_IF


PreviousState := THIS^.State;

CASE THIS^.State OF 
	
	E_ALARM_STATE.ACTIVE_UNACK:
	
		CASE THIS^.Config.Acknowledge OF
			
			E_ALARM_ACK_TYPE.ONLY_ACK:
				THIS^.State := E_ALARM_STATE.INACTIVE;
				
			E_ALARM_ACK_TYPE.ACK_OR_RESET:
				THIS^.State := E_ALARM_STATE.INACTIVE;
			
			E_ALARM_ACK_TYPE.ACK_AFTER_RESET:
				;
				
			ELSE
				THIS^.State := E_ALARM_STATE.ACTIVE_ACK;
			
		END_CASE;

	E_ALARM_STATE.INACTIVE_UNACK:
		
		THIS^.State := E_ALARM_STATE.INACTIVE;
					
	ELSE
		;
		
END_CASE;

IF THIS^.State <> PreviousState THEN
	THIS^.Handler.RegisterAlarm(Alarm := THIS^, Prefix := '', Update := TRUE);
END_IF;

Acknowledge REF= THIS^;
END_METHOD

METHOD PUBLIC AcknowledgeNoUpdate : REFERENCE TO FB_ALARM
VAR_INPUT
END_VAR
VAR
	PreviousState : E_ALARM_STATE;
END_VAR
{warning disable C0371}

// Checking the VAR_IN_OUT reference, leave the current method in case of invalid reference
IF NOT __ISVALIDREF(THIS^.Handler) THEN
     RETURN;
END_IF


PreviousState := THIS^.State;

CASE THIS^.State OF 
	
	E_ALARM_STATE.ACTIVE_UNACK:
	
		CASE THIS^.Config.Acknowledge OF
			
			E_ALARM_ACK_TYPE.ONLY_ACK:
				THIS^.State := E_ALARM_STATE.INACTIVE;
				
			E_ALARM_ACK_TYPE.ACK_OR_RESET:
				THIS^.State := E_ALARM_STATE.INACTIVE;
			
			E_ALARM_ACK_TYPE.ACK_AFTER_RESET:
				;
				
			ELSE
				THIS^.State := E_ALARM_STATE.ACTIVE_ACK;
			
		END_CASE;

	E_ALARM_STATE.INACTIVE_UNACK:
		
		THIS^.State := E_ALARM_STATE.INACTIVE;
					
	ELSE
		;
		
END_CASE;

IF THIS^.State <> PreviousState THEN
	THIS^.Handler.RegisterAlarm(Alarm := THIS^, Prefix := '', Update := FALSE);
END_IF;

AcknowledgeNoUpdate REF= THIS^;
END_METHOD

METHOD PUBLIC Activate : REFERENCE TO FB_ALARM
VAR_INPUT
END_VAR
VAR
	PreviousState : E_ALARM_STATE;
END_VAR
{warning disable C0371}

// Checking the VAR_IN_OUT reference, leave the current method in case of invalid reference
IF NOT __ISVALIDREF(THIS^.Handler) THEN
     RETURN;
END_IF


PreviousState := THIS^.State;

CASE THIS^.State OF 
	
	E_ALARM_STATE.ACTIVE_ACK:
		// Keeps the state as active and acknowledged
		;
			
	ELSE
		// Any other state will turn it into active and unacknowledged
		THIS^.State := E_ALARM_STATE.ACTIVE_UNACK;
		
END_CASE;

IF THIS^.State <> PreviousState THEN
	THIS^.Handler.RegisterAlarm(Alarm := THIS^, Prefix := '', Update := TRUE);
END_IF;

Activate REF= THIS^;
END_METHOD

PROPERTY PUBLIC IsActive : BOOL
GET
IsActive := THIS^.State = E_ALARM_STATE.ACTIVE_ACK OR THIS^.State = E_ALARM_STATE.ACTIVE_UNACK;
END_GET
END_PROPERTY

METHOD PUBLIC Reset : REFERENCE TO FB_ALARM
VAR_INPUT
END_VAR
VAR
	PreviousState : E_ALARM_STATE;
END_VAR
{warning disable C0371}

// Checking the VAR_IN_OUT reference, leave the current method in case of invalid reference
IF NOT __ISVALIDREF(THIS^.Handler) THEN
     RETURN;
END_IF


PreviousState := THIS^.State;

CASE THIS^.State OF 
	
	E_ALARM_STATE.ACTIVE_UNACK:
	
		CASE THIS^.Config.Acknowledge OF
			
			E_ALARM_ACK_TYPE.ONLY_RESET:
				THIS^.State := E_ALARM_STATE.INACTIVE;
				
			E_ALARM_ACK_TYPE.ACK_OR_RESET:
				THIS^.State := E_ALARM_STATE.INACTIVE;
				
			ELSE
				THIS^.State := E_ALARM_STATE.INACTIVE_UNACK;
			
		END_CASE;
		
	E_ALARM_STATE.ACTIVE_ACK:
		THIS^.State := E_ALARM_STATE.INACTIVE;
			
	ELSE
		;
		
END_CASE;

IF THIS^.State <> PreviousState THEN
	THIS^.Handler.RegisterAlarm(Alarm := THIS^, Prefix := '', Update := TRUE);
END_IF;

Reset REF= THIS^;
END_METHOD

END_FUNCTION_BLOCK

// ---- Base/Alarms/Repository/FB_ALARM_REPOSITORY.TcPOU
FUNCTION_BLOCK PUBLIC FB_ALARM_REPOSITORY EXTENDS FBA_ALARM_HANDLER;
VAR_IN_OUT
	Alarms : ARRAY[*] OF FB_ALARM_INSTANCE;
	VisuAlarms : ARRAY[*] OF TYP_VISU_ALARM;
END_VAR
VAR_INPUT
	AcknowledgeAll : BOOL;
END_VAR
VAR_OUTPUT
END_VAR
VAR
END_VAR

IF AcknowledgeAll THEN
	THIS^._acknowledgeAll();
	AcknowledgeAll := FALSE;
END_IF;

METHOD PRIVATE _acknowledgeAll;
VAR
	i: DINT;
END_VAR
FOR i:= LOWER_BOUND(THIS^.Alarms, 1) TO UPPER_BOUND(THIS^.Alarms, 1) DO
	IF __ISVALIDREF(THIS^.Alarms[i].Alarm) THEN
		THIS^.Alarms[i].Alarm.AcknowledgeNoUpdate();
	END_IF;
END_FOR;

THIS^.UpdateAlarms().SortAlarms().PopulateVisuAlarms();
END_METHOD

{attribute 'monitoring' := 'call'}
PROPERTY PUBLIC ActiveAlarms : USINT
GET
VAR
	i : DINT;
	cnt : DINT;
END_VAR
cnt := 0;

FOR i:= LOWER_BOUND(THIS^.VisuAlarms, 1) TO UPPER_BOUND(THIS^.VisuAlarms, 1) DO
	IF THIS^.VisuAlarms[i].State <> 'INACTIVE' THEN
		cnt := cnt + 1;
	END_IF
END_FOR;

ActiveAlarms := DINT_TO_USINT(cnt);
END_GET
END_PROPERTY

METHOD PRIVATE AddAlarm : REFERENCE TO FB_ALARM_REPOSITORY
VAR_INPUT
	AlarmInstance : FB_ALARM_INSTANCE;
END_VAR
VAR
	i : DINT;
END_VAR
FOR i:= LOWER_BOUND(THIS^.Alarms, 1) TO UPPER_BOUND(THIS^.Alarms, 1) DO
	IF NOT __ISVALIDREF(THIS^.Alarms[i].Alarm) THEN
		THIS^.Alarms[i] := AlarmInstance;
		EXIT;
	END_IF;
END_FOR;

AddAlarm REF= THIS^;
END_METHOD

METHOD PRIVATE CreateAlarmInstance : FB_ALARM_INSTANCE
VAR_INPUT
	Alarm : REFERENCE TO FB_ALARM;
	Prefix : STRING;
END_VAR
VAR
	AlarmInstance : FB_ALARM_INSTANCE;
END_VAR
AlarmInstance.Alarm REF= Alarm;
AlarmInstance.ActivationDateTime := BASE.DateTime.GetCurrentDateTime();
AlarmInstance.Config := Alarm.Config;
AlarmInstance.Config.Name := CONCAT(Prefix, Alarm.Config.Name);
AlarmInstance.State := Alarm.State;

CreateAlarmInstance := AlarmInstance;
END_METHOD

METHOD PRIVATE IsAlarmPresent : BOOL
VAR_INPUT
	Alarm : REFERENCE TO FB_ALARM;
END_VAR
VAR
	i : DINT;
	lwr : DINT;
	upr : DINT;
END_VAR
IsAlarmPresent := FALSE;

lwr := LOWER_BOUND(THIS^.Alarms, 1);
upr := UPPER_BOUND(THIS^.Alarms, 1);
FOR i:= lwr TO upr DO
	IF ADR(THIS^.Alarms[i].Alarm) = ADR(Alarm) AND __ISVALIDREF(THIS^.Alarms[i].Alarm) THEN
		IsAlarmPresent := TRUE;
		EXIT;
	END_IF;
END_FOR;
END_METHOD

PROPERTY PROTECTED NullAlarmInstance : FB_ALARM_INSTANCE
GET
VAR
	AlarmInstance : FB_ALARM_INSTANCE;
END_VAR
AlarmInstance.ActivationDateTime := DWORD_TO_DT(0);

AlarmInstance.Alarm REF= 0;

AlarmInstance.Config.Acknowledge := E_ALARM_ACK_TYPE.ONLY_ACK;
AlarmInstance.Config.Code := 0;
AlarmInstance.Config.MultiInstance := FALSE;
AlarmInstance.Config.Name := '';
AlarmInstance.Config.Priority := 0;

AlarmInstance.State := E_ALARM_STATE.INACTIVE;

NullAlarmInstance := AlarmInstance;
END_GET
END_PROPERTY

METHOD PRIVATE PopulateVisuAlarms : REFERENCE TO FB_ALARM_REPOSITORY
VAR_INPUT
END_VAR

VAR
	i: DINT;
END_VAR
FOR i:= LOWER_BOUND(THIS^.Alarms, 1) TO UPPER_BOUND(THIS^.Alarms, 1) DO
	IF i >= LOWER_BOUND(THIS^.VisuAlarms, 1) AND i <= UPPER_BOUND(THIS^.VisuAlarms, 1) THEN
		THIS^.VisuAlarms[i] := THIS^.Alarms[i].VisuAlarm;
	END_IF;
END_FOR;

PopulateVisuAlarms REF= THIS^;
END_METHOD

METHOD RegisterAlarm : REFERENCE TO FBA_ALARM_HANDLER
VAR_INPUT
	Alarm	: REFERENCE TO FB_ALARM;
	Prefix	: STRING := '';
	Update : BOOL;
END_VAR

VAR
	i: DINT;
END_VAR
IF NOT THIS^.IsAlarmPresent(Alarm := Alarm) OR (Alarm.Config.MultiInstance AND Alarm.State = E_ALARM_STATE.ACTIVE_UNACK) THEN
	THIS^.AddAlarm(AlarmInstance := THIS^.CreateAlarmInstance(Alarm := Alarm, Prefix := Prefix));
END_IF;

IF Update THEN
	THIS^.UpdateAlarms().SortAlarms().PopulateVisuAlarms();
END_IF;

RegisterAlarm REF= THIS^;
END_METHOD

METHOD PRIVATE SortAlarms : REFERENCE TO FB_ALARM_REPOSITORY
VAR_INPUT
END_VAR

VAR
	i: DINT;
	j: DINT;
	Found : BOOL;
END_VAR
FOR i:= LOWER_BOUND(THIS^.Alarms, 1) TO UPPER_BOUND(THIS^.Alarms, 1) DO
	IF NOT __ISVALIDREF(THIS^.Alarms[i].Alarm) THEN
		Found := FALSE;
		FOR j:= i TO UPPER_BOUND(THIS^.Alarms, 1) DO
			IF __ISVALIDREF(THIS^.Alarms[j].Alarm) THEN
				THIS^.Alarms[i] := THIS^.Alarms[j];
				THIS^.Alarms[j] := THIS^.NullAlarmInstance;
				Found := TRUE;
				EXIT;
			END_IF;
		END_FOR;
		IF NOT Found THEN
			EXIT;
		END_IF;
	END_IF;
END_FOR;

SortAlarms REF= THIS^;
END_METHOD

METHOD PRIVATE UpdateAlarms : REFERENCE TO FB_ALARM_REPOSITORY
VAR_INPUT
END_VAR

VAR
	i: DINT;
END_VAR
FOR i:= LOWER_BOUND(THIS^.Alarms, 1) TO UPPER_BOUND(THIS^.Alarms, 1) DO
	THIS^.Alarms[i].Update();
	
	IF THIS^.Alarms[i].State <> E_ALARM_STATE.ACTIVE_ACK AND THIS^.Alarms[i].State <> E_ALARM_STATE.ACTIVE_UNACK AND THIS^.Alarms[i].State <> E_ALARM_STATE.INACTIVE_UNACK THEN
		THIS^.Alarms[i] := THIS^.NullAlarmInstance;
	END_IF;
END_FOR;

UpdateAlarms REF= THIS^;
END_METHOD

END_FUNCTION_BLOCK

// ---- Base/Alarms/Repository/FB_ALARM_INSTANCE.TcPOU
FUNCTION_BLOCK PUBLIC FB_ALARM_INSTANCE
VAR_INPUT
	Alarm : REFERENCE TO FB_ALARM;
	Config : TYP_ALARM_CONFIG;
	State : E_ALARM_STATE;
END_VAR
VAR_OUTPUT
END_VAR
VAR
	_actDT : DT;
END_VAR

PROPERTY PUBLIC ActivationDateTime : DT
GET
ActivationDateTime := THIS^._actDT;
END_GET
SET
THIS^._actDT :=	ActivationDateTime;
END_SET
END_PROPERTY

METHOD PUBLIC Update : REFERENCE TO FB_ALARM_INSTANCE
VAR_INPUT
END_VAR
IF __ISVALIDREF(THIS^.Alarm) THEN
	THIS^.State := THIS^.Alarm.State;
END_IF;

Update REF= THIS^;
END_METHOD

PROPERTY PUBLIC VisuAlarm : TYP_VISU_ALARM
GET
VAR
	Alarm : TYP_VISU_ALARM;
END_VAR
Alarm.Code := THIS^.Config.Code;
Alarm.Priority := THIS^.Config.Priority;
Alarm.Message := THIS^.Config.Name;
Alarm.Name := THIS^.Config.Name;
Alarm.Timestamp := THIS^.ActivationDateTime;
Alarm.State := TO_STRING(THIS^.State);

VisuAlarm := Alarm;
END_GET
END_PROPERTY

END_FUNCTION_BLOCK

// ---- Base/BASE.TcPOU
PROGRAM BASE
VAR
	DateTime : FB_DATETIME;
	Strings : FB_STRINGS;
END_VAR

DateTime();
Strings();

END_PROGRAM

// ---- Base/DateTime/FB_DATETIME.TcPOU
FUNCTION_BLOCK PUBLIC FB_DATETIME
VAR_INPUT
END_VAR
VAR_OUTPUT
END_VAR
VAR
END_VAR

METHOD PUBLIC GetCurrentDateTime : DT
VAR_INPUT
END_VAR
VAR
	SystemTime    : GETSYSTEMTIME;
	timeAsFileTime  : T_FILETIME;
	timeAsDT        : DT;
END_VAR
SystemTime( timeLoDW =>timeAsFileTime.dwLowDateTime , timeHiDW =>timeAsFileTime.dwHighDateTime );
GetCurrentDateTime := FILETIME_TO_DT( timeAsFileTime );
END_METHOD

METHOD PUBLIC GetTimeDiff : TIME
VAR_INPUT
	In1 : TIME;
	In2 : TIME;
END_VAR
GetTimeDiff := In2 - In1;
END_METHOD

METHOD PUBLIC GetTimeSince : TIME
VAR_INPUT
	In : TIME;
END_VAR
GetTimeSince := TIME() - In;
END_METHOD

END_FUNCTION_BLOCK

// ---- Base/String/FB_STRINGS.TcPOU
FUNCTION_BLOCK PUBLIC FB_STRINGS
VAR_INPUT
END_VAR
VAR_OUTPUT
END_VAR
VAR
END_VAR

METHOD PUBLIC IsNumeric : BOOL
VAR_INPUT
	In : STRING;
END_VAR
VAR
	i : USINT;
	NewString : STRING;
	Pos : INT;
END_VAR
IF In = '' THEN
	IsNumeric := FALSE;
ELSE
	NewString := In;
	IF FIND(NewString, '-') = 1 THEN
		NewString := DELETE(NewString, 1, 1);
	END_IF;
	FOR i := 0 TO 9 DO
		WHILE TRUE DO
			Pos := FIND(NewString, TO_STRING(i));
			IF Pos <> 0 THEN
				NewString := DELETE(NewString, 1, Pos);
			ELSE
				EXIT;
			END_IF;
		END_WHILE;
	END_FOR;
	IsNumeric := LEN(NewString) = 0;
END_IF
END_METHOD

END_FUNCTION_BLOCK

// ---- Main/PurgeN2/FB_PURGE_N2.TcPOU
FUNCTION_BLOCK FB_PURGE_N2 EXTENDS FBA_SEQUENCE
VAR_INPUT

END_VAR
VAR_IN_OUT
	Control : TYP_PURGE_N2_CONTROL;
	Parameter: TYP_PURGE_N2_PARAMETER;
END_VAR
VAR_OUTPUT
	Status : TYP_PURGE_N2_STATUS;
END_VAR
VAR
	AlarmHandler : FB_ALARM_HANDLER;
	fbPurgeN2GeneralError : FB_ALARM;
	bInit : BOOL;
	bReset : BOOL;
	bTestalarm : BOOL;
	bTestReset : BOOL;
	bTestAcknowledge : BOOL;
	fbPurgeN2Device : FB_N2_DEVICE;
	State : E_N2_STATES;
END_VAR

//Open valves
//Start purging
//Check if purging time reached
//Repeat x times
//Close valves
//Done := TRUE
IF bInit THEN
	THIS^.Initialize();
	bInit := FALSE;
END_IF

IF bReset THEN
	THIS^.Reset();
	bReset := FALSE;
END_IF

AlarmHandler(Prefix:='PURGE_N2', Repository:=AlarmRepository);
fbPurgeN2GeneralError.Config.Acknowledge := E_ALARM_ACK_TYPE.ACK_AND_RESET;
fbPurgeN2GeneralError.Config.Name := 'PURGE_N2_GENERAL_ERROR';
fbPurgeN2GeneralError.Config.Priority := 3;
fbPurgeN2GeneralError.Config.Code := 1000;
fbPurgeN2GeneralError(Handler := AlarmHandler);

fbPurgeN2Device.AlarmConfig.Name := 'N2_DEVICE';
fbPurgeN2Device.AlarmConfig.Handler REF= AlarmHandler;
fbPurgeN2Device();

//Example how alarms work
IF bTestalarm THEN
	fbPurgeN2GeneralError.Activate();
ELSIF bTestReset THEN
	fbPurgeN2GeneralError.Reset();
ELSIF bTestAcknowledge THEN
	fbPurgeN2GeneralError.Acknowledge();
END_IF

_state(State := State, AlarmHandler := AlarmHandler, StateAsString := TO_STRING(State));

METHOD PUBLIC  Initialize : REFERENCE TO FBA_SEQUENCE
VAR_INPUT
END_VAR
END_METHOD

METHOD PUBLIC  Reset : REFERENCE TO FBA_SEQUENCE
VAR_INPUT
END_VAR
END_METHOD

END_FUNCTION_BLOCK

// ---- Base/States/FBA_SEQUENCE.TcPOU
FUNCTION_BLOCK ABSTRACT FBA_SEQUENCE
VAR_IN_OUT
	AlarmRepository : FB_ALARM_REPOSITORY;
END_VAR
VAR_INPUT
END_VAR
VAR_OUTPUT
	Initialized : BOOL;
END_VAR
VAR
	_state : FB_STATE_MACHINE;
END_VAR

METHOD PUBLIC ABSTRACT Initialize : REFERENCE TO FBA_SEQUENCE
VAR_INPUT
END_VAR
END_METHOD

METHOD PUBLIC ABSTRACT Reset : REFERENCE TO FBA_SEQUENCE
VAR_INPUT
END_VAR
END_METHOD

END_FUNCTION_BLOCK

// ---- Main/PurgeN2/FB_N2_DEVICE.TcPOU
FUNCTION_BLOCK FB_N2_DEVICE
VAR_INPUT
	AlarmConfig : TYP_ALARM_DEVICE_CONFIG;
END_VAR
VAR_OUTPUT
END_VAR
VAR
	bTestalarm : BOOL;
	bTestReset : BOOL;
	bTestAcknowledge : BOOL;
	fbPurgeN2DeviceError : FB_ALARM;
END_VAR

fbPurgeN2DeviceError.Config.Acknowledge := E_ALARM_ACK_TYPE.ACK_AND_RESET;
fbPurgeN2DeviceError.Config.Name := CONCAT(AlarmConfig.Name, '*PURGE_N2_GENERAL_ERROR');
fbPurgeN2DeviceError.Config.Priority := 3;
fbPurgeN2DeviceError(Handler := AlarmConfig.Handler);

IF bTestalarm THEN
	fbPurgeN2DeviceError.Activate();
ELSIF bTestReset THEN
	fbPurgeN2DeviceError.Reset();
ELSIF bTestAcknowledge THEN
	fbPurgeN2DeviceError.Acknowledge();
END_IF

END_FUNCTION_BLOCK

// ---- Main/PressureControl/FB_PRES_CNTRL.TcPOU
FUNCTION_BLOCK FB_PRES_CNTRL
VAR_INPUT

END_VAR
VAR_IN_OUT
	Control : TYP_PRES_CNTRL_CONTROL;
	Parameter: TYP_PRES_CNTRL_PARAMETER;
END_VAR
VAR_OUTPUT
	Status : TYP_PRES_CNTRL_STATUS;
END_VAR
VAR
END_VAR

END_FUNCTION_BLOCK

// ---- Base/Basic/FB_RS_TRIG.TcPOU
FUNCTION_BLOCK PUBLIC FB_RS_TRIG
VAR_INPUT
	CLK : BOOL;
END_VAR
VAR_OUTPUT
	Q : BOOL; // pos edge
	QS : BOOL; // pos edge set
END_VAR
VAR
	Trig : R_TRIG;
END_VAR

Trig(CLK := CLK, Q => Q);
IF Trig.Q THEN
	QS := TRUE;
END_IF;

METHOD PUBLIC Reset : REFERENCE TO FB_RS_TRIG
VAR_INPUT
END_VAR
THIS^.QS := FALSE;

Reset REF= THIS^;
END_METHOD

END_FUNCTION_BLOCK

// ---- Base/Files/FB_FIND_FILES.TcPOU
FUNCTION_BLOCK PUBLIC FB_FIND_FILES
VAR_IN_OUT
	Filenames : ARRAY[*] OF STRING;
END_VAR
VAR_INPUT
	Filter : STRING;
	Execute : BOOL;
	Abort : BOOL;
END_VAR
VAR_OUTPUT
	Busy : BOOL;
	Done : BOOL;
	Error : BOOL;
END_VAR
VAR
	State : INT;
	i : DINT;
	FindFile : FB_EnumFindFileEntry;
END_VAR

CASE State OF 
	0: 
		Busy := FALSE;
		IF Execute THEN
			Done := FALSE;
			Error := FALSE;
			Busy := TRUE;
			Execute := FALSE;
			FindFile.eCmd := eEnumCmd_First;
			FindFile.sPathName := Filter;
			
			FOR i := LOWER_BOUND(Filenames, 1) TO UPPER_BOUND(Filenames, 1) DO
				Filenames[i] := '';
			END_FOR;
			
			i := LOWER_BOUND(Filenames, 1);
			State := 10;
		END_IF;
		
	10:
		IF Abort THEN
            Abort      := FALSE;
            FindFile.eCmd := eEnumCmd_Abort;
        END_IF
        FindFile(bExecute := FALSE);
        FindFile(bExecute := TRUE);
        State := 20;
		
	20:
		FindFile(bExecute := FALSE);
        IF NOT FindFile.bBusy THEN
            IF NOT FindFile.bError THEN
                IF NOT FindFile.bEOE AND i <= UPPER_BOUND(Filenames, 1) THEN
					Filenames[i] := FindFile.stFindFile.sFileName;
					i := i + 1;
					FindFile.eCmd := eEnumCmd_Next;
					State := 10;
                ELSE
					Done := TRUE;
                    State := 0;
                END_IF
            ELSE
                Error := TRUE;
                State     := 0;
            END_IF
        END_IF
END_CASE;

END_FUNCTION_BLOCK

// ---- Base/Math/FC_SCALE.TcPOU
FUNCTION FC_SCALE : REAL
VAR_INPUT
	In : REAL;
	Conf : TYP_SCALE_CONF;
END_VAR
VAR
END_VAR

FC_SCALE := ((Conf.OutMax - Conf.OutMin) / (Conf.InMax - Conf.InMin) * In) + Conf.OutMin;

END_FUNCTION

// ---- Base/Motion/DC/DcMotor/FB_DC_MOTOR.TcPOU
FUNCTION_BLOCK FB_DC_MOTOR
VAR_IN_OUT
	Hardware : TYP_DC_MOTOR_HW;
END_VAR
VAR_INPUT
END_VAR
VAR_OUTPUT
	Status : TYP_DC_MOTOR_STATUS;
END_VAR
VAR
	_cmdRun : BOOL;
	_cmdChangeDir : BOOL;
	_cmdNewDir : BOOL;
	PreDelay : TON;
	PostDelay : TON;
END_VAR

IF _cmdRun AND NOT _cmdChangeDir THEN
	IF Hardware.Out.Direction AND Hardware.In.LimitWP THEN
		_cmdRun := FALSE;
	ELSIF NOT Hardware.Out.Direction AND Hardware.In.LimitHP THEN
		_cmdRun := FALSE;
	END_IF;
END_IF;

PreDelay(IN := _cmdChangeDir, PT := T#500MS);
PostDelay(IN := PreDelay.Q, PT := T#500MS);

IF _cmdChangeDir THEN
	THIS^.Hardware.Out.Run := FALSE;
	
	IF PostDelay.Q THEN
		_cmdChangeDir := FALSE;
	ELSIF PreDelay.Q THEN
		THIS^.Hardware.Out.Direction := _cmdNewDir;
	END_IF;
ELSE
	THIS^.Hardware.Out.Run := _cmdRun;
END_IF;

Status.ReachedHP := Hardware.In.LimitHP;
Status.ReachedWP := Hardware.In.LimitWP;

METHOD PUBLIC Run : REFERENCE TO FB_DC_MOTOR
VAR_INPUT
END_VAR
_cmdRun := TRUE;

Run REF= THIS^;
END_METHOD

METHOD PUBLIC SetDirection : REFERENCE TO FB_DC_MOTOR
VAR_INPUT
	Direction : BOOL; // FALSE = forward, TRUE = reverse
END_VAR
VAR
	
END_VAR
_cmdChangeDir := TRUE;
_cmdNewDir := Direction;

SetDirection REF= THIS^;
END_METHOD

METHOD PUBLIC Stop : REFERENCE TO FB_DC_MOTOR
VAR_INPUT
END_VAR
_cmdRun := FALSE;

Stop REF= THIS^;
END_METHOD

END_FUNCTION_BLOCK

// ---- Base/Motion/DC/Faulhaber_SC/FB_FAULHABER_SC.TcPOU
FUNCTION_BLOCK PUBLIC FB_FAULHABER_SC
VAR_IN_OUT
	Hardware : TYP_FAULHABER_SC_HW;
END_VAR
VAR_INPUT
	AlarmConfig : TYP_ALARM_DEVICE_CONFIG;
	Control : TYP_FAULHABER_SC_CTRL;
END_VAR
VAR_OUTPUT
	Error : BOOL;
END_VAR
VAR
	FaultAlarm : FB_ALARM;
END_VAR

FaultAlarm.Config.Acknowledge := E_ALARM_ACK_TYPE.ACK_AND_RESET;
FaultAlarm.Config.Name := CONCAT(AlarmConfig.Name, '_DRIVE_FAULT');
FaultAlarm(Handler := AlarmConfig.Handler);

IF Hardware.In.Fault THEN
	FaultAlarm.Activate();
END_IF;

Error := Hardware.In.Fault;

IF Control.Run AND Control.Enable THEN
	Hardware.Out.Speed := ABS(Control.Speed);
	Hardware.Out.Direction := Control.Speed >= 0;
ELSE
	Hardware.Out.Speed := 0;
END_IF;

END_FUNCTION_BLOCK

// ---- Base/Pneumatics/FB_VALVE_TIMEOUT_ALARM.TcPOU
FUNCTION_BLOCK PUBLIC FB_VALVE_TIMEOUT_ALARM
VAR_IN_OUT
	Handler : FB_ALARM_HANDLER;
	Config : TYP_VALVE_TIMEOUT_ALARM_CONF;
END_VAR
VAR_INPUT
	Condition : BOOL;
END_VAR
VAR_OUTPUT
	Error : BOOL;
END_VAR
VAR
	_alarm : FB_ALARM;
	Timer : TON;
	PosEdge : R_TRIG;
	NegEdge : F_TRIG;
END_VAR

Timer(IN := Condition, PT := Config.Delay);

PosEdge(CLK := Timer.Q);
NegEdge(CLK := Timer.Q);

_alarm(Handler := Handler);

IF PosEdge.Q AND Config.Enable THEN
	_alarm.Activate();
END_IF;

IF NegEdge.Q THEN
	_alarm.Reset();
END_IF;

Error := Timer.Q;

PROPERTY PUBLIC Alarm : REFERENCE TO FB_ALARM
GET
Alarm REF= THIS^._alarm;
END_GET
END_PROPERTY

END_FUNCTION_BLOCK

// ---- Base/Pneumatics/VacuumGen/FB_VAC_GEN.TcPOU
FUNCTION_BLOCK PUBLIC FB_VAC_GEN
VAR_IN_OUT
	Hardware : TYP_VAC_GEN_HW;
END_VAR
VAR_INPUT
	Control : TYP_VAC_GEN_CTRL;
	Config : TYP_VAC_GEN_CONF;
	AlarmConfig : TYP_ALARM_DEVICE_CONFIG;
END_VAR
VAR_OUTPUT
	Status : TYP_VAC_GEN_STATUS;
END_VAR
VAR
	CmdActivate : BOOL;
	CmdRelease : BOOL;
	VacAlarm : FB_ALARM;
	VacAlarmTime : TON;
	VacAlarmEdge : R_TRIG;
	ServiceEdge : R_TRIG;
	ReleaseTime : TIME;
END_VAR

VacAlarm.Config.Acknowledge := E_ALARM_ACK_TYPE.ACK_AND_RESET;
VacAlarm.Config.Name := CONCAT(AlarmConfig.Name, '*NO_VAC');
VacAlarm(Handler := AlarmConfig.Handler);
VacAlarmTime(IN := CmdActivate AND NOT Status.ReachedVac, PT := Config.Alarm.Timeout);
VacAlarmEdge(CLK := VacAlarmTime.Q);

IF VacAlarmEdge.Q AND Config.Alarm.Enable THEN
	VacAlarm.Activate();
END_IF;

IF NOT CmdActivate AND VacAlarm.IsActive THEN
	VacAlarm.Reset();
END_IF;

ServiceEdge(CLK := Control.ServiceEnable);

IF ServiceEdge.Q THEN // Remember command when entering service mode to avoid unpredictable movements
	Control.ServiceActivate := CmdActivate;
	Control.ServiceRelease := CmdRelease;
END_IF;

IF Control.ServiceEnable THEN
	CmdActivate := Control.ServiceActivate;
	CmdRelease := Control.ServiceRelease;
END_IF;

Hardware.Out.EnableVac := CmdActivate;
Hardware.Out.ReleaseVac := CmdRelease;

Status.ReachedVac := Hardware.In.ReachedVac;
Status.Error := VacAlarm.IsActive;

IF NOT Control.ServiceEnable THEN
	IF Status.ReachedVac AND NOT Config.Permanent THEN
		Hardware.Out.EnableVac := FALSE;
	END_IF;
	
	IF CmdRelease AND TIME() - ReleaseTime > T#1S THEN
		CmdRelease := FALSE;
	END_IF;
END_IF;

METHOD PUBLIC Activate : REFERENCE TO FB_VAC_GEN
VAR_INPUT
END_VAR
IF THIS^.Control.Enable AND THIS^.Control.EnableActivate THEN
	CmdActivate := TRUE;
	CmdRelease := FALSE;
END_IF;

Activate REF= THIS^;
END_METHOD

METHOD PUBLIC Release : REFERENCE TO FB_VAC_GEN
VAR_INPUT
END_VAR
IF THIS^.Control.Enable AND THIS^.Control.EnableRelease THEN
	CmdActivate := FALSE;
	CmdRelease := TRUE;
	ReleaseTime := TIME();
END_IF;

Release REF= THIS^;
END_METHOD

METHOD PUBLIC Reset : REFERENCE TO FB_VAC_GEN
VAR_INPUT
END_VAR

CmdActivate := FALSE;
CmdRelease := FALSE;


Reset REF= THIS^;
END_METHOD

END_FUNCTION_BLOCK

// ---- Base/Pneumatics/Valve53/FB_VALVE_53.TcPOU
FUNCTION_BLOCK FB_VALVE_53
VAR_IN_OUT
	Hardware : TYP_VALVE_53_HW;
END_VAR
VAR_INPUT
	Control : TYP_VALVE_53_CTRL;
	Config : TYP_VALVE_53_CONF;
	AlarmConfig : TYP_ALARM_DEVICE_CONFIG;
END_VAR
VAR_OUTPUT
	Status : TYP_VALVE_53_STATUS;
END_VAR
VAR
	CmdHP : BOOL;
	CmdWP : BOOL;
	TimeoutHP : FB_VALVE_TIMEOUT_ALARM;
	TimeoutWP : FB_VALVE_TIMEOUT_ALARM;
	TimeoutHP_WP : FB_VALVE_TIMEOUT_ALARM;
	SensorlessDelayHP : TON;
	SensorlessDelayWP : TON;
	ServiceEdge : R_TRIG;
END_VAR

TimeoutHP.Alarm.Config.Acknowledge := E_ALARM_ACK_TYPE.ACK_AND_RESET;
TimeoutHP.Alarm.Config.Name := CONCAT(AlarmConfig.Name, '*HP_ALARM');
TimeoutHP.Condition := NOT Hardware.In.ReachedHP AND Hardware.Out.CmdHP;
TimeoutHP(Config := Config.HP.Timeout, Handler := AlarmConfig.Handler);

TimeoutWP.Alarm.Config.Acknowledge := E_ALARM_ACK_TYPE.ACK_AND_RESET;
TimeoutWP.Alarm.Config.Name := CONCAT(AlarmConfig.Name, '*WP_ALARM');
TimeoutWP.Condition := NOT Hardware.In.ReachedWP AND Hardware.Out.CmdWP;
TimeoutWP(Config := Config.WP.Timeout, Handler := AlarmConfig.Handler);

TimeoutHP_WP.Alarm.Config.Acknowledge := E_ALARM_ACK_TYPE.ACK_AND_RESET;
TimeoutHP_WP.Alarm.Config.Name := CONCAT(AlarmConfig.Name, '*HP_WP_ALARM');
TimeoutHP_WP.Condition := Hardware.In.ReachedHP AND Hardware.In.ReachedWP;
TimeoutHP_WP(Config := Config.HP_WP, Handler := AlarmConfig.Handler);

ServiceEdge(CLK := Control.ServiceEnable);

IF ServiceEdge.Q THEN // Remember command when entering service mode to avoid unpredictable movements
	Control.ServiceHP := CmdHP;
	Control.ServiceWP := CmdWP;
END_IF;

IF Control.ServiceEnable THEN
	CmdHP := Control.ServiceHP;
	CmdWP := Control.ServiceWP;
END_IF;

Hardware.Out.CmdHP := CmdHP;
Hardware.Out.CmdWP := CmdWP;

IF Control.BlockOutputs THEN
	Hardware.Out.CmdHP := FALSE;
	Hardware.Out.CmdWP := FALSE;
END_IF;

SensorlessDelayHP(IN := CmdHP AND Config.HP.Sensorless, PT := Config.HP.SensorlessDelay);
SensorlessDelayWP(IN := CmdWP AND Config.WP.Sensorless, PT := Config.WP.SensorlessDelay);

Status.ReachedHP := ((Hardware.In.ReachedHP AND NOT Hardware.In.ReachedWP) AND NOT Config.HP.Sensorless) OR SensorlessDelayHP.Q;
Status.ReachedWP := ((Hardware.In.ReachedWP AND NOT Hardware.In.ReachedHP) AND NOT Config.WP.Sensorless) OR SensorlessDelayWP.Q;

// Turn off physical output in case of non-permanent position mode
IF NOT Control.ServiceEnable THEN
	IF Status.ReachedHP AND NOT Config.HP.Permanent THEN
		Hardware.Out.CmdHP := FALSE;
	END_IF;
	
	IF Status.ReachedWP AND NOT Config.WP.Permanent THEN
		Hardware.Out.CmdWP := FALSE;
	END_IF;
END_IF;

Status.Error := TimeoutHP.Alarm.IsActive OR TimeoutWP.Alarm.IsActive OR TimeoutHP_WP.Alarm.IsActive;

METHOD PUBLIC ActivateHP : REFERENCE TO FB_VALVE_53
VAR_INPUT
END_VAR
IF THIS^.Control.Enable AND THIS^.Control.EnableHP THEN
	CmdHP := TRUE;
	CmdWP := FALSE;
END_IF;


ActivateHP REF= THIS^;
END_METHOD

METHOD PUBLIC ActivateWP : REFERENCE TO FB_VALVE_53
VAR_INPUT
END_VAR
IF THIS^.Control.Enable AND THIS^.Control.EnableWP THEN
	CmdWP := TRUE;
	CmdHP := FALSE;
END_IF;


ActivateWP REF= THIS^;
END_METHOD

PROPERTY PUBLIC IO : REFERENCE TO TYP_VALVE_53_HW
GET
{warning disable C0371}

IF __ISVALIDREF(THIS^.Hardware) THEN
     IO REF= THIS^.Hardware;
END_IF
END_GET
END_PROPERTY

METHOD PUBLIC Release : REFERENCE TO FB_VALVE_53
VAR_INPUT
END_VAR
IF THIS^.Control.Enable THEN
	CmdWP := FALSE;
	CmdHP := FALSE;
END_IF;

Release REF= THIS^;
END_METHOD

METHOD PUBLIC Reset : REFERENCE TO FB_VALVE_53
VAR_INPUT
END_VAR
THIS^.CmdHP := FALSE;
THIS^.CmdWP := FALSE;
THIS^.Control.ServiceEnable := FALSE;
THIS^.Control.ServiceHP := FALSE;
THIS^.Control.ServiceWP := FALSE;

Reset REF= THIS^;
END_METHOD

END_FUNCTION_BLOCK

// ---- Base/Robotics/UR/Profinet/FB_UR_PN.TcPOU
FUNCTION_BLOCK PUBLIC FB_UR_PN
VAR_IN_OUT
	Hardware : TYP_HW_UR_PN;
END_VAR
VAR
	_pnIO : FB_UR_PN_IO;
	_state : TYP_UR_PN_STATE;
	_tcp : TYP_UR_PN_TCP;
END_VAR

_pnIO(Hardware := THIS^.Hardware);

METHOD PUBLIC ReadBitRegister : BOOL
VAR_INPUT
	Register : USINT;
END_VAR
VAR
	RegByte : USINT;
	RegBit : USINT;
	RefByte : BYTE;
END_VAR
{warning disable C0371}

IF __ISVALIDREF(THIS^.Hardware) THEN
	RegByte := DINT_TO_USINT(TRUNC(USINT_TO_REAL(Register) / 8.0));
	RegBit := Register MOD 8;
	
	IF RegByte <= 7 THEN
		RefByte := THIS^.Hardware.In.T2OURBitReg[RegByte];
	END_IF;
	
	ReadBitRegister := FC_GET_BIT_IN_BYTE(BitToGet := RegBit, RefByte := ADR(RefByte));
END_IF;
END_METHOD

METHOD PUBLIC ReadFloatRegister : REAL
VAR_INPUT
	Register : USINT;
END_VAR
VAR
	RegByte : USINT;
	PtrByte : POINTER TO BYTE;
	ReturnReal : REAL;
END_VAR
{warning disable C0371}

IF __ISVALIDREF(THIS^.Hardware) THEN
	RegByte := Register * 4;
	
	IF RegByte <= 23 THEN
		PtrByte := ADR(THIS^.Hardware.In.T2OURFloatReg[RegByte]);
	END_IF;
	
	FC_FLIP_DWORD(In := PtrByte, Out := ADR(ReturnReal));
	
	ReadFloatRegister := ReturnReal;
END_IF;
END_METHOD

METHOD PUBLIC ReadIntRegister : DINT
VAR_INPUT
	Register : USINT;
END_VAR
VAR
	RegByte : USINT;
	PtrByte : POINTER TO BYTE;
	ReturnDint : DINT;
END_VAR
{warning disable C0371}

IF __ISVALIDREF(THIS^.Hardware) THEN
	RegByte := 4 * Register;
	
	IF RegByte <= 23 THEN
		PtrByte := ADR(THIS^.Hardware.In.T2OURIntReg[RegByte]);
	END_IF;
	
	FC_FLIP_DWORD(In := PtrByte, Out := ADR(ReturnDint));
	ReadIntRegister := ReturnDint;
END_IF;
END_METHOD

PROPERTY PUBLIC RobotIO : REFERENCE TO FB_UR_PN_IO
GET
RobotIO REF= THIS^._pnIO;
END_GET
END_PROPERTY

PROPERTY PUBLIC State : REFERENCE TO TYP_UR_PN_STATE
GET
{warning disable C0371}

IF __ISVALIDREF(THIS^.Hardware) THEN
	_state.MajVersion := THIS^.Hardware.In.T2OURState[0];
	_state.MinVersion := THIS^.Hardware.In.T2OURState[1];
	_state.RobotMode := BYTE_TO_INT(THIS^.Hardware.In.T2OURState[4]);
	_state.RTMs := THIS^.Hardware.In.T2OURState[5];
	_state.RTMs := THIS^.Hardware.In.T2OURState[5];
	_state.RTMm := THIS^.Hardware.In.T2OURState[8];
	_state.RTMh := THIS^.Hardware.In.T2OURState[9];
	FC_FLIP_WORD(In := ADR(THIS^.Hardware.In.T2OURState[6]), Out := ADR(_state.RTMms));
	FC_FLIP_WORD(In := ADR(THIS^.Hardware.In.T2OURState[10]), Out := ADR(_state.RTMd));
	FC_FLIP_DWORD(In := ADR(THIS^.Hardware.In.T2OURState[12]), Out := ADR(_state.RobotCurrent));
	_state.Power := THIS^.Hardware.In.T2OURState[16].0;
	_state.ProgramRunning := THIS^.Hardware.In.T2OURState[16].1;
	_state.TeachButton := THIS^.Hardware.In.T2OURState[16].2;
	_state.PowerButton := THIS^.Hardware.In.T2OURState[16].3;
	_state.NormalMode := THIS^.Hardware.In.T2OURState[28].0;
	_state.ReducedMode := THIS^.Hardware.In.T2OURState[28].1;
	_state.ProtectiveStopped := THIS^.Hardware.In.T2OURState[28].2;
	_state.RecoveryMode := THIS^.Hardware.In.T2OURState[28].3;
	_state.SafeguardStop := THIS^.Hardware.In.T2OURState[28].4;
	_state.SystemEmergencyStopped := THIS^.Hardware.In.T2OURState[28].5;
	_state.RobotEmergencyStopped := THIS^.Hardware.In.T2OURState[28].6;
	_state.EmergencyStopped := THIS^.Hardware.In.T2OURState[28].7;
	_state.Violation := THIS^.Hardware.In.T2OURState[29].0;
	_state.Faulted := THIS^.Hardware.In.T2OURState[29].1;
	_state.SafetyStopped := THIS^.Hardware.In.T2OURState[29].2;
END_IF;


State REF= _state;
END_GET
END_PROPERTY

PROPERTY PUBLIC TCP : REFERENCE TO TYP_UR_PN_TCP
GET
{warning disable C0371}

IF __ISVALIDREF(THIS^.Hardware) THEN
	FC_FLIP_DWORD(In := ADR(THIS^.Hardware.In.T2OURTCP[0]), Out := ADR(THIS^._tcp.Position.X));
	FC_FLIP_DWORD(In := ADR(THIS^.Hardware.In.T2OURTCP[4]), Out := ADR(THIS^._tcp.Position.Y));
	FC_FLIP_DWORD(In := ADR(THIS^.Hardware.In.T2OURTCP[8]), Out := ADR(THIS^._tcp.Position.Z));
	
	FC_FLIP_DWORD(In := ADR(THIS^.Hardware.In.T2OURTCP[12]), Out := ADR(THIS^._tcp.PositionR.X));
	FC_FLIP_DWORD(In := ADR(THIS^.Hardware.In.T2OURTCP[16]), Out := ADR(THIS^._tcp.PositionR.Y));
	FC_FLIP_DWORD(In := ADR(THIS^.Hardware.In.T2OURTCP[20]), Out := ADR(THIS^._tcp.PositionR.Z));
	
	FC_FLIP_DWORD(In := ADR(THIS^.Hardware.In.T2OURTCP[24]), Out := ADR(THIS^._tcp.Velocity.X));
	FC_FLIP_DWORD(In := ADR(THIS^.Hardware.In.T2OURTCP[28]), Out := ADR(THIS^._tcp.Velocity.Y));
	FC_FLIP_DWORD(In := ADR(THIS^.Hardware.In.T2OURTCP[32]), Out := ADR(THIS^._tcp.Velocity.Z));
	
	FC_FLIP_DWORD(In := ADR(THIS^.Hardware.In.T2OURTCP[36]), Out := ADR(THIS^._tcp.VelocityR.X));
	FC_FLIP_DWORD(In := ADR(THIS^.Hardware.In.T2OURTCP[40]), Out := ADR(THIS^._tcp.VelocityR.Y));
	FC_FLIP_DWORD(In := ADR(THIS^.Hardware.In.T2OURTCP[44]), Out := ADR(THIS^._tcp.VelocityR.Z));
	
	FC_FLIP_DWORD(In := ADR(THIS^.Hardware.In.T2OURTCP[48]), Out := ADR(THIS^._tcp.Force.X));
	FC_FLIP_DWORD(In := ADR(THIS^.Hardware.In.T2OURTCP[52]), Out := ADR(THIS^._tcp.Force.Y));
	FC_FLIP_DWORD(In := ADR(THIS^.Hardware.In.T2OURTCP[56]), Out := ADR(THIS^._tcp.Force.Z));
	
	FC_FLIP_DWORD(In := ADR(THIS^.Hardware.In.T2OURTCP[60]), Out := ADR(THIS^._tcp.Torque.X));
	FC_FLIP_DWORD(In := ADR(THIS^.Hardware.In.T2OURTCP[64]), Out := ADR(THIS^._tcp.Torque.Y));
	FC_FLIP_DWORD(In := ADR(THIS^.Hardware.In.T2OURTCP[68]), Out := ADR(THIS^._tcp.Torque.Z));
	
	FC_FLIP_DWORD(In := ADR(THIS^.Hardware.In.T2OURTCP[72]), Out := ADR(THIS^._tcp.ForceScalar));
END_IF;


TCP REF= _tcp;
END_GET
END_PROPERTY

METHOD PUBLIC WriteBitRegister
VAR_INPUT
	Register : USINT;
	Value : BOOL;
END_VAR
VAR
	RegByte : USINT;
	RegBit : USINT;
	RefByte : REFERENCE TO BYTE;
END_VAR
{warning disable C0371}

IF __ISVALIDREF(THIS^.Hardware) THEN
	RegByte := DINT_TO_USINT(TRUNC(USINT_TO_REAL(Register) / 8.0));
	RegBit := Register MOD 8;
	
	IF RegByte <= 3 THEN
		RefByte REF= THIS^.Hardware.Out.O2TURGenReg1[RegByte];
	ELSIF RegByte <= 7 THEN
		RefByte REF= THIS^.Hardware.Out.O2TURGenReg2[RegByte-4];
	END_IF;
	
	FC_SET_BIT_IN_BYTE(BitToSet := RegBit, RefByte := ADR(RefByte), Value := Value);
END_IF;
END_METHOD

METHOD PUBLIC WriteFloatRegister
VAR_INPUT
	Register : USINT;
	Value : REAL;
END_VAR
VAR
	RegByte : USINT;
	PtrByte : POINTER TO BYTE;
END_VAR
{warning disable C0371}

IF __ISVALIDREF(THIS^.Hardware) THEN
	RegByte := (Register MOD 12) * 4;
	
	IF Register <= 11 THEN
		PtrByte := ADR(THIS^.Hardware.Out.O2TURGenReg1[RegByte + 52]);
	ELSIF Register <= 23 THEN
		PtrByte := ADR(THIS^.Hardware.Out.O2TURGenReg2[RegByte + 52]);
	END_IF;
	
	FC_FLIP_DWORD(In := ADR(Value), Out := PtrByte);
END_IF;
END_METHOD

METHOD PUBLIC WriteIntRegister
VAR_INPUT
	Register : USINT;
	Value : DINT;
END_VAR
VAR
	RegByte : USINT;
	PtrByte : POINTER TO BYTE;
END_VAR
{warning disable C0371}

IF __ISVALIDREF(THIS^.Hardware) THEN
	RegByte := 4 + (4 * Register);
	
	IF RegByte <= 11 THEN
		PtrByte := ADR(THIS^.Hardware.Out.O2TURGenReg1[RegByte]);
	ELSIF RegByte <= 23 THEN
		PtrByte := ADR(THIS^.Hardware.Out.O2TURGenReg2[RegByte]);
	END_IF;
	
	FC_FLIP_DWORD(In := ADR(Value), PtrByte);
END_IF;
END_METHOD

END_FUNCTION_BLOCK

// ---- Base/Robotics/UR/Profinet/FB_UR_PN_IO.TcPOU
FUNCTION_BLOCK PUBLIC FB_UR_PN_IO
VAR_IN_OUT
	Hardware : TYP_HW_UR_PN;
END_VAR
VAR_INPUT
END_VAR
VAR_OUTPUT
END_VAR
VAR
	_speedSlider : REAL;
END_VAR

// Future versions should include digital and analog IO too, wasn't necessary in this application

IF THIS^.Hardware.Out.O2TURIO[0].0 THEN // Speed slider mask to false when written
	IF _speedSlider = THIS^.SpeedSlider THEN
		THIS^.Hardware.Out.O2TURIO[0].0 := FALSE; 
	END_IF;
END_IF;

PROPERTY PUBLIC PumpVoltage : REAL
GET
VAR
	TempReal: REAL;
END_VAR
{warning disable C0371}

IF __ISVALIDREF(THIS^.Hardware) THEN

	FC_FLIP_DWORD(In := ADR(THIS^.Hardware.In.T2OURIO[16]), Out := ADR(TempReal));
	PumpVoltage := TempReal;
	
END_IF;
END_GET
END_PROPERTY

PROPERTY PUBLIC SpeedSlider : REAL
GET
VAR
	TempReal : REAL;
END_VAR
{warning disable C0371}

IF __ISVALIDREF(THIS^.Hardware) THEN

	FC_FLIP_DWORD(In := ADR(THIS^.Hardware.In.T2OURState[20]), Out := ADR(TempReal));
	SpeedSlider := TempReal;
	
END_IF;
END_GET
SET
{warning disable C0371}

IF __ISVALIDREF(THIS^.Hardware) THEN

	IF NOT THIS^.Hardware.Out.O2TURIO[0].0 THEN // Speed slider mask
		FC_FLIP_DWORD(In := ADR(SpeedSlider), Out := ADR(THIS^.Hardware.Out.O2TURIO[4]));
		_speedSlider := SpeedSlider;
		THIS^.Hardware.Out.O2TURIO[0].0 := TRUE; 
	END_IF
	
END_IF;
END_SET
END_PROPERTY

END_FUNCTION_BLOCK

// ---- Base/Twiddlers/FC_FLIP_DWORD.TcPOU
FUNCTION FC_FLIP_DWORD
VAR_INPUT
	In : POINTER TO BYTE;
	Out : POINTER TO BYTE;
END_VAR
VAR
	ByteArray : ARRAY[0..3] OF BYTE;
	ReturnArray : ARRAY[0..3] OF BYTE;
END_VAR

MEMCPY(srcAddr := In, destAddr := ADR(ByteArray), n := 4);

ReturnArray[0] := ByteArray[3];
ReturnArray[1] := ByteArray[2];
ReturnArray[2] := ByteArray[1];
ReturnArray[3] := ByteArray[0];

MEMCPY(srcAddr := ADR(ReturnArray), destAddr := Out, n := 4);

END_FUNCTION

// ---- Base/Twiddlers/FC_GET_BIT_IN_BYTE.TcPOU
FUNCTION FC_GET_BIT_IN_BYTE : BOOL
VAR_INPUT
	RefByte : POINTER TO BYTE;
	BitToGet : USINT;
END_VAR
VAR
END_VAR

CASE BitToGet OF
	
	0:
		FC_GET_BIT_IN_BYTE := BIT_TO_BOOL(RefByte^.0);
	1:
		FC_GET_BIT_IN_BYTE := BIT_TO_BOOL(RefByte^.1);
	2:
		FC_GET_BIT_IN_BYTE := BIT_TO_BOOL(RefByte^.2);
	3:
		FC_GET_BIT_IN_BYTE := BIT_TO_BOOL(RefByte^.3);
	4:
		FC_GET_BIT_IN_BYTE := BIT_TO_BOOL(RefByte^.4);
	5:
		FC_GET_BIT_IN_BYTE := BIT_TO_BOOL(RefByte^.5);
	6:	
		FC_GET_BIT_IN_BYTE := BIT_TO_BOOL(RefByte^.6);
	7:
		FC_GET_BIT_IN_BYTE := BIT_TO_BOOL(RefByte^.7);
		
END_CASE;

END_FUNCTION

// ---- Base/Twiddlers/FC_FLIP_WORD.TcPOU
FUNCTION FC_FLIP_WORD
VAR_INPUT
	In : POINTER TO BYTE;
	Out : POINTER TO BYTE;
END_VAR
VAR
	ByteArray : ARRAY[0..1] OF BYTE;
	ReturnArray : ARRAY[0..1] OF BYTE;
END_VAR

MEMCPY(srcAddr := In, destAddr := ADR(ByteArray), n := 2);

ReturnArray[0] := ByteArray[1];
ReturnArray[1] := ByteArray[0];

MEMCPY(srcAddr := ADR(ReturnArray), destAddr := Out, n := 2);

END_FUNCTION

// ---- Base/Twiddlers/FC_SET_BIT_IN_BYTE.TcPOU
FUNCTION FC_SET_BIT_IN_BYTE : BOOL
VAR_INPUT
	Value : BOOL;
	RefByte : POINTER TO BYTE;
	BitToSet : USINT;
END_VAR
VAR
END_VAR

CASE BitToSet OF
	
	0:
		RefByte^.0 := Value;
	1:
		RefByte^.1 := Value;
	2:
		RefByte^.2 := Value;
	3:
		RefByte^.3 := Value;
	4:
		RefByte^.4 := Value;
	5:
		RefByte^.5 := Value;
	6:	
		RefByte^.6 := Value;
	7:
		RefByte^.7 := Value;
		
END_CASE;

END_FUNCTION

// ---- Base/Serial/FB_EL6001_LINE_CTRL.TcPOU
FUNCTION_BLOCK FB_EL6001_LINE_CTRL
VAR_IN_OUT
	EL6001 : TYP_HW_EL6001;

END_VAR
VAR_INPUT
END_VAR
VAR_OUTPUT
END_VAR
VAR
	SerialLineControl : SerialLineControl;
	Buffer : TYP_SERIAL_DATA;
END_VAR

SerialLineControl.Mode := ComSerialLineMode_t.SERIALLINEMODE_EL6_22B;
SerialLineControl.pComIn := ADR(EL6001.In.COM);
SerialLineControl.pComOut := ADR(EL6001.Out.COM);
SerialLineControl.SizeComIn := UINT_TO_INT(SIZEOF(EL6001.In.COM));
SerialLineControl(RxBuffer := Buffer.RxData, TxBuffer := Buffer.TxData);

PROPERTY PUBLIC RxBuffer : REFERENCE TO COMbuffer
GET
RxBuffer REF= THIS^.Buffer.RxData;
END_GET
END_PROPERTY

PROPERTY PUBLIC TxBuffer : REFERENCE TO COMbuffer
GET
TxBuffer REF= THIS^.Buffer.TxData;
END_GET
END_PROPERTY

END_FUNCTION_BLOCK

// ---- Base/Serial/FB_EL6001_RS232.TcPOU
FUNCTION_BLOCK PUBLIC FB_EL6001_RS232
VAR_IN_OUT
	LineCtrl : FB_EL6001_LINE_CTRL;
END_VAR
VAR_INPUT
	Send : BOOL;
END_VAR
VAR_OUTPUT
END_VAR
VAR
	ReceiveString : ReceiveString255;
	SendString : SendString255;
	RecvStr : STRING[255];
	SendStr : STRING[255];
END_VAR

ReceiveString(RXbuffer := LineCtrl.RxBuffer, ReceivedString := RecvStr, Timeout := T#1S);

IF Send THEN
	SendString(TXbuffer := LineCtrl.TxBuffer, SendString := SendStr);
	IF NOT SendString.Busy THEN
		Send := FALSE;
	END_IF;
END_IF;

END_FUNCTION_BLOCK

// ---- Base/Signalling/BannerK50/FB_BANNER_K50.TcPOU
FUNCTION_BLOCK PUBLIC FB_BANNER_K50
VAR_IN_OUT
	Hardware : TYP_BAN_K50_HW;
END_VAR
VAR_INPUT
END_VAR
VAR_OUTPUT
	ButtonPressed : BOOL;
	ButtonPosEdge : BOOL;
	ButtonNegEdge : BOOL;
END_VAR
VAR
	PosTrig : R_TRIG;
	NegTrig : F_TRIG;
END_VAR

ButtonPressed := Hardware.In.ButtonPressed;

PosTrig(CLK := ButtonPressed, Q => ButtonPosEdge);
NegTrig(CLK := ButtonPressed, Q => ButtonNegEdge);

METHOD PUBLIC SetGreenLight : REFERENCE TO FB_BANNER_K50
VAR_INPUT
END_VAR
{warning disable C0371}

// Checking the VAR_IN_OUT reference, leave the current method in case of invalid reference
IF NOT __ISVALIDREF(THIS^.Hardware) THEN
     RETURN;
END_IF

THIS^.Hardware.Out.Green := TRUE;

SetGreenLight REF= THIS^;
END_METHOD

METHOD PUBLIC SetRedLight : REFERENCE TO FB_BANNER_K50
VAR_INPUT
END_VAR
{warning disable C0371}

// Checking the VAR_IN_OUT reference, leave the current method in case of invalid reference
IF NOT __ISVALIDREF(THIS^.Hardware) THEN
     RETURN;
END_IF


THIS^.Hardware.Out.Red := TRUE;

SetRedLight REF= THIS^;
END_METHOD

METHOD PUBLIC SetYellowLight : REFERENCE TO FB_BANNER_K50
VAR_INPUT
END_VAR
{warning disable C0371}

// Checking the VAR_IN_OUT reference, leave the current method in case of invalid reference
IF NOT __ISVALIDREF(THIS^.Hardware) THEN
     RETURN;
END_IF


THIS^.Hardware.Out.Yellow := TRUE;

SetYellowLight REF= THIS^;
END_METHOD

METHOD PUBLIC TurnOffLights : REFERENCE TO FB_BANNER_K50
VAR_INPUT
END_VAR
{warning disable C0371}

// Checking the VAR_IN_OUT reference, leave the current method in case of invalid reference
IF NOT __ISVALIDREF(THIS^.Hardware) THEN
     RETURN;
END_IF


THIS^.Hardware.Out.Green := FALSE;
THIS^.Hardware.Out.Yellow := FALSE;
THIS^.Hardware.Out.Red := FALSE;

TurnOffLights REF= THIS^;
END_METHOD

END_FUNCTION_BLOCK

// ---- Base/Signalling/RGB/FB_RGB_LED.TcPOU
FUNCTION_BLOCK PUBLIC FB_RGB_LED
VAR_IN_OUT
	Hardware : TYP_RGB_LED_HW;
END_VAR
VAR_INPUT
END_VAR
VAR_OUTPUT
END_VAR
VAR
END_VAR

METHOD PUBLIC SetRGB : REFERENCE TO FB_RGB_LED
VAR_INPUT
	Red : USINT;
	Green : USINT;
	Blue : USINT;
END_VAR
{warning disable C0371}

// Checking the VAR_IN_OUT reference, leave the current method in case of invalid reference
IF NOT __ISVALIDREF(THIS^.Hardware) THEN
     RETURN;
END_IF

THIS^.Hardware.Red.Out.PWM := REAL_TO_INT((USINT_TO_REAL(Red) / 255) * 32767);
THIS^.Hardware.Green.Out.PWM := REAL_TO_INT((USINT_TO_REAL(Green) / 255) * 32767);
THIS^.Hardware.Blue.Out.PWM := REAL_TO_INT((USINT_TO_REAL(Blue) / 255) * 32767);
END_METHOD

END_FUNCTION_BLOCK

// ---- Base/States/FB_SEQUENCE_VISU.TcPOU
FUNCTION_BLOCK PUBLIC FB_SEQUENCE_VISU
VAR_IN_OUT
	Sequence : FBA_SEQUENCE;
END_VAR
VAR_INPUT
	Start : BOOL;
	Stop : BOOL;
	Reset : BOOL;
	Initialize : BOOL;
	HmiState : STRING;
END_VAR
VAR_OUTPUT
END_VAR
VAR
END_VAR

IF Initialize THEN
	Sequence.Initialize();
	Initialize := FALSE;
END_IF;

IF Reset THEN
	Sequence.Reset();
	Reset := FALSE;
END_IF;

IF Start THEN
	Sequence._state.Start();
	Start := FALSE;
END_IF;

IF Stop THEN
	Sequence._state.Stop();
	Stop := FALSE;
END_IF;

END_FUNCTION_BLOCK

// ---- Base/Twiddlers/FC_MEMCPY_FLIP_WORD.TcPOU
FUNCTION FC_MEMCPY_FLIP_WORD : BOOL
VAR_IN_OUT
	Source : ARRAY[*] OF BYTE;
END_VAR
VAR_INPUT
	Dest : POINTER TO BYTE;
END_VAR
VAR
	ArrLen : UDINT;
	NewArray : POINTER TO BYTE;
	i : DINT;
	Overflow : DINT;
END_VAR

ArrLen := DINT_TO_UDINT((UPPER_BOUND(Source,1) - LOWER_BOUND(Source,1)) + 1);

NewArray := __NEW(BYTE, ArrLen);
Overflow := UDINT_TO_DINT(ArrLen MOD 4);

FOR i := LOWER_BOUND(Source,1) TO UPPER_BOUND(Source,1) BY 4 DO
	IF i < (UPPER_BOUND(Source,1) - Overflow) THEN
		NewArray[i] := Source[i + 3];
		NewArray[i + 1] := Source[i + 2];
		NewArray[i + 2] := Source[i + 1];
		NewArray[i + 3] := Source[i];
	ELSE
		NewArray[i] := Source[i];
	END_IF;
END_FOR;

MEMCPY(Dest, NewArray, ArrLen);

__DELETE(NewArray);

END_FUNCTION

// ---- Base/Twiddlers/FC_MEMCPY_SWAP_BYTE.TcPOU
FUNCTION FC_MEMCPY_SWAP_BYTE : BOOL
VAR_IN_OUT
	Source : ARRAY[*] OF BYTE;
END_VAR
VAR_INPUT
	Dest : POINTER TO BYTE;
END_VAR
VAR
	ArrLen : UDINT;
	NewArray : POINTER TO BYTE;
	i : DINT;
END_VAR

ArrLen := DINT_TO_UDINT((UPPER_BOUND(Source,1) - LOWER_BOUND(Source,1)) + 1);

NewArray := __NEW(BYTE, ArrLen);

FOR i := LOWER_BOUND(Source,1) TO UPPER_BOUND(Source,1) BY 2 DO
	IF i < UPPER_BOUND(Source,1) THEN
		NewArray[i] := Source[i + 1];
		NewArray[i + 1] := Source[i];
	ELSE
		NewArray[i] := Source[i];
	END_IF;
END_FOR;

MEMCPY(Dest, NewArray, ArrLen);

__DELETE(NewArray);

END_FUNCTION

// ---- Base/Twiddlers/FC_MEMCPY_SWAP_WORD.TcPOU
FUNCTION FC_MEMCPY_SWAP_WORD : BOOL
VAR_IN_OUT
	Source : ARRAY[*] OF BYTE;
END_VAR
VAR_INPUT
	Dest : POINTER TO BYTE;
END_VAR
VAR
	ArrLen : UDINT;
	NewArray : POINTER TO BYTE;
	i : DINT;
	Overflow : DINT;
END_VAR

ArrLen := DINT_TO_UDINT((UPPER_BOUND(Source,1) - LOWER_BOUND(Source,1)) + 1);

NewArray := __NEW(BYTE, ArrLen);
Overflow := UDINT_TO_DINT(ArrLen MOD 4);

FOR i := LOWER_BOUND(Source,1) TO UPPER_BOUND(Source,1) BY 4 DO
	IF i < (UPPER_BOUND(Source,1) - Overflow) THEN
		NewArray[i] := Source[i + 2];
		NewArray[i + 1] := Source[i + 3];
		NewArray[i + 2] := Source[i];
		NewArray[i + 3] := Source[i + 1];
	ELSE
		NewArray[i] := Source[i];
	END_IF;
END_FOR;

MEMCPY(Dest, NewArray, ArrLen);

__DELETE(NewArray);

END_FUNCTION
